// TIA Portal V20 export
// export: Created 2025-12-01T14:56:46.3467956Z, ExportSetting None, DisplayName Totally Integrated Automation Portal, DisplayVersion V20 Update 3, DisplayName TIA Portal Openness, DisplayVersion V20 Update 3, DisplayName TIA Portal Version Control Interface, DisplayVersion V20 Update 3, DisplayName STEP 7 Professional, DisplayVersion V20 Update 3, DisplayName STEP 7 Safety, DisplayVersion V20 Update 2, DisplayName WinCC Basic/Comfort/Advanced, DisplayVersion V20 Update 3, DisplayName WinCC Professional, DisplayVersion V20 Update 3, DisplayName WinCC Unified, DisplayVersion V20 Update 3
FUNCTION_BLOCK "FB263_M_FSS_Maquetas"   // FB263, LAD
TITLE = Control del Ramal de Salidas
{ S7_Optimized_Access := 'FALSE' }
AUTHOR : TE_FSS
NAME : 20160509
VERSION : 3.4
// stored: AutoNumber false, SetENOAutomatically false
   VAR_INPUT
      Mesa : UInt;   // Existe Tension en la Mesa
      Error_Tx : Bool;   // Error en el Tx
      EnTension : Bool;   // Mesa de la FB
      Termico_Tx : Bool;   // Proteccion del Tx
      pHsMx_MQ1 : Bool;   // pHs de la Mesa >> En MQ1
      pHsMx_MQ2 : Bool;   // pHs de la Mesa >> En MQ2
      Avance_Tx : Bool;   // Avance del Tx
      TP1_Arriba : Bool;   // TP1 Arriba. Nota Movimiento E1 >> S3
      TP1_Abajo : Bool;   // TP1 Abajo. Nota Movimiento E1 >> S3
      EnMovimiento_TP1 : Bool;   // En movimiento el TP1
      MQ1_Arriba : Bool;   // MQ1 Arriba >> 1º UT de la Mesa
      MQ1_Abajo : Bool;   // MQ1 Abajo >> 1º UT de la Mesa
      EnMovimiento_MQ1 : Bool;   // MQ1 EnMovimiento >> 1º UT de la Mesa
      MQ2_Arriba : Bool;   // MQ2 Arriba >> 2º UT de la Mesa
      MQ2_Abajo : Bool;   // MQ2 Abajo >> 2º UT de la Mesa
      EnMovimiento_MQ2 : Bool;   // MQ2 EnMovimiento >> 2º UT de la Mesa
      MAnt_DescargaAct : Bool;   // E1 >> Mesa Anterior DescargaAct
      AVTF_MAnt_Mx_MQ1 : Bool;   // E1 >> Mesa Anterior AVTF
      AVTF_MAnt_Mx_MQ1_2 : Bool;   // E1 >> Mesa Anterior AVTF
      P_Mens_MAnt_Mx : Bool;   // E1 >> Mesa Anterior P_Mens
      PTF_Mx_MSig : Bool;   // S3 >> Mesa Siguiente PTF
      FTF_Mx_MSig : Bool;   // S3 >> Mesa Siguiente FTF
      MSig_CargaAct : Bool;
      Mx_ControlUTs : Bool;   // Config >> Control de UT en Mesa
      F_EnvMens_Mx : Bool;   // Fin de Envio de Mensaje
      OrdSal_MQ1 : Bool;   // Orden de Salida de MQ1
      OrdSal_MQ2 : Bool;   // Orden de Salida de MQ2
      OrdSal_MQ1_2 : Bool;   // Orden de Salida de MQ1 y MQ2
      V_CNT_pHsMx : Int := 400;   // Valor de Presencia
      V_CNT_pHsMx_FTF : Int := 200;   // Valor para activar FTF. Nota: < = V_CNT_pHsMx.
      V_CNTSeg_pHsMx : Int := 2000;   // Valor de Seguriadad para Presencia
      V_CNT_ApHsMx : Int := 200;   // Valor de Ausencia
      V_CNTSeg_ApHsMx : Int := 2000;   // Valor de Seguriadad para Ausencia
      V_CNT_Simultaneo : Int := 2000;   // Valor de Simultaneo
      V_EstabilidadCarga : Time := T#200MS;   // Valor de Estabilidad de la Carga
      V_RetardoBajarMAQ : Time := T#200MS;   // Valor de Retardo de Bajada de las Maquetas
      V_TOut_Tx_Mx : Int := 7000;   // TimeOut de Entrada por E1
      V_TOut_TP : Int := 3000;   // TimeOut de Tope
      V_TOut_MQ : Int := 3000;   // TimeOut de Maqueta
      V_CNT_PerdidapHs : Int := 1000;   // CNT de Perdida de pHs
   END_VAR
   VAR_OUTPUT
      P_EnvMens_PMx : Bool;   // Permiso de Enviar Mensaje de Presencia
      P_RecepOK_Mx : Bool;   // Recepcion OK
      PTF_MAnt_Mx : Bool;   // E1 >> Mesa Anterior PTF
      FTF_MAnt_Mx : Bool;   // E1 >> Mesa Anterior FTF
      AVTF_Mx_MSig_MQ1 : Bool;   // S3 >> Mesa Siguiente AVTF
      AVTF_Mx_MSig_MQ2 : Bool;   // S3 >> Mesa Siguiente AVTF
      AVTF_Mx_MSig_MQ1_2 : Bool;   // S3 >> Mesa Siguiente AVTF
      P_Mens_Mx_MSig : Bool;   // S3 >> Mesa Siguiente P_Mens
   END_VAR
   VAR
      Mx_ET00 : Bool;
      Mx_ET01 : Bool;
      Mx_ET02 : Bool;
      Mx_ET06 : Bool;
      Mx_ET07 : Bool;
      Mx_ET08 : Bool;
      Mx_ET09 : Bool;
      Mx_ET10 : Bool;
      Mx_ET11 : Bool;
      Mx_ET12 : Bool;
      Mx_ET110 : Bool;
      Mx_ET111 : Bool;
      Mx_ET50 : Bool;
      Mx_ET51 : Bool;
      Mx_ET150 : Bool;
      Mx_ET151 : Bool;
      SinUTs_EnMesa : Bool;   // Control UTs En Mesa >> Sin UTs
      DoblePeque_EnMesa : Bool;   // Control UTs En Mesa >> Caja Doble Pequeña
      UT01Peque_EnMesa : Bool;   // Control UTs En Mesa >> UT01 Caja Pequeña
      UT02Peque_EnMesa : Bool;   // Control UTs En Mesa >> UT02 Caja Pequeña
      OrdSalida_OK : Bool;   // Control UTs En Mesa >> Validar Orden de Salida
      Selec_Entrada : Bool;   // Select Entrada de Mesa Anterior
      Selec_Salida_MQ1 : Bool;   // Select Salida de MQ1
      Selec_Salida_MQ2 : Bool;   // Select Salida de MQ2
      Selec_Salida_MQ1_2 : Bool;   // Select Salida de MQ1 y MQ2
      AVTF_MAnt_Mx : Bool;   // Interna >> Aviso de Entrada
      AVTF_Mx_MSig : Bool;   // Interna >> Aviso de Salida
      SaliendoCarga : Bool;   // Interna >> Realizando Salida de la Mesa
      PosMQ_OK : Bool;   // Interna >> Pos. de Maquetas OK
      Simultaneo_Mx : Bool;   // Activo Simultaneo E1
      ProtocoloIniciado : Bool;   // Iniciado el Envio del Mensaje de Presencia
      CNT_pHsMx_FTF_OK : Bool;   // Enviar ya FTF
      STAT_EnvMens_PMx : Bool;   // Interna >> Envio del Mensaje de Presencia
      STAT_FTF_MAnt_Mx : Bool;   // Interna >> FTF de MAnt >> Mx
      MA_Subir_MQ1 : Bool;
      MA_Bajar_MQ1 : Bool;
      MA_Subir_MQ2 : Bool;
      MA_Bajar_MQ2 : Bool;
      TMP_EstabilidadCarga { S7_SetPoint := 'True'} : TON_TIME;   // TMP de Estabilidad de la Carga En la Entrada
      TMP_RetardoBajada_MQ1 { S7_SetPoint := 'True'} : TON_TIME;   // TMP de Retardo de Bajada de la MQ1
      TMP_RetardoBajada_MQ2 { S7_SetPoint := 'True'} : TON_TIME;   // TMP de Retardo de Bajada de la MQ2
      CNT_pHsMx { S7_SetPoint := 'True'} : "FB910_CNT_UHS";   // CNT de la Presencia
      CNTSeg_pHsMx { S7_SetPoint := 'True'} : "FB910_CNT_UHS";   // CNT de Seguridad de la Presencia
      CNT_ApHsMx { S7_SetPoint := 'True'} : "FB910_CNT_UHS";   // CNT de la Ausencia
      CNTSeg_ApHsMx { S7_SetPoint := 'True'} : "FB910_CNT_UHS";   // CNT de Seguridad de la Ausencia
      CNT_Simultaneo { S7_SetPoint := 'True'} : "FB910_CNT_UHS";   // CNT de Simultaneo
      TMP_EnTension { S7_SetPoint := 'True'} : "FB910_CNT_UHS";
      TOut_Av_Mx { S7_SetPoint := 'True'} : "FB910_CNT_UHS";   // Time Out de Entrada de E1
      TOut_Subir_TP { S7_SetPoint := 'True'} : "FB910_CNT_UHS";   // Time Out de Subida del TP
      TOut_Bajar_TP { S7_SetPoint := 'True'} : "FB910_CNT_UHS";   // Time Out de Bajada del TP
      TOut_Subir_MQ { S7_SetPoint := 'True'} : "FB910_CNT_UHS";
      TOut_Bajar_MQ { S7_SetPoint := 'True'} : "FB910_CNT_UHS";
      CNT_PerdidapHs { S7_SetPoint := 'True'} : "FB910_CNT_UHS";   // CNT de Perdida de pHs
   END_VAR
   VAR_TEMP
      EstadoZona : "EstadoZona";   // Estado de Zona de la Mesa
      EstadoVI : "EstadosMesa";   // Estado del Vehiculo Inteliguente de la Mesa
      ConfigFB : "UDT_ConfigFB";   // Configuracion de la FB de la Mesa
      V_Protrusion : Int;
      Aux_ET00 : Bool;
   END_VAR
   VAR_TEMP   // added for the SCL form of the ladder/FBD networks
      _w1 : Bool;
   END_VAR
BEGIN

REGION Network 1: INICIALIZAR - Recoger las Variables de Estado de la Mesa
   // Se recoge - Estado_CBx
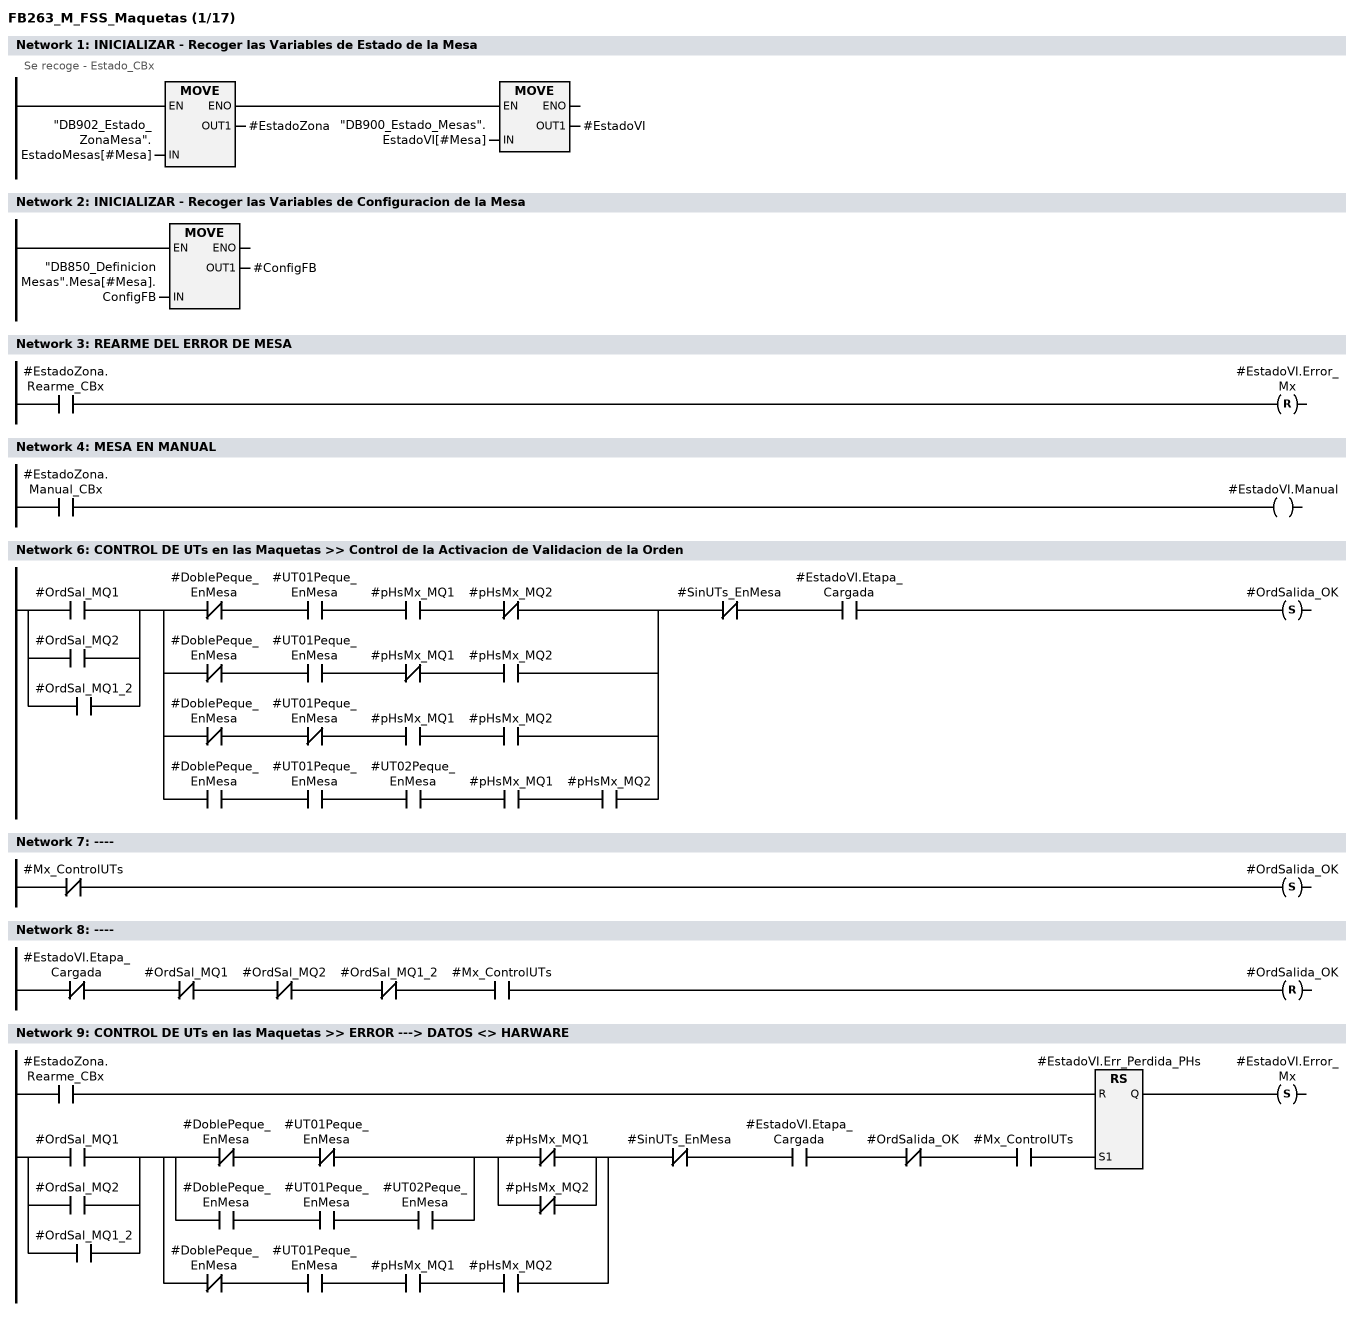
   RUNG wire#powerrail
      Move(in := "DB902_Estado_ZonaMesa".EstadoMesas[#Mesa], out1 => #EstadoZona)
      Move(in := "DB900_Estado_Mesas".EstadoVI[#Mesa], out1 => #EstadoVI)
   END_RUNG
   // the same network as SCL:
   #EstadoZona := "DB902_Estado_ZonaMesa".EstadoMesas[#Mesa];
   #EstadoVI := "DB900_Estado_Mesas".EstadoVI[#Mesa];
END_REGION

REGION Network 2: INICIALIZAR - Recoger las Variables de Configuracion de la Mesa
   RUNG wire#powerrail
      Move(in := "DB850_DefinicionMesas".Mesa[#Mesa].ConfigFB, out1 => #ConfigFB)
   END_RUNG
   // the same network as SCL:
   #ConfigFB := "DB850_DefinicionMesas".Mesa[#Mesa].ConfigFB;
END_REGION

REGION Network 3: REARME DEL ERROR DE MESA
   RUNG wire#powerrail
      Contact( #EstadoZona.Rearme_CBx )
      R_Coil( #EstadoVI.Error_Mx )
   END_RUNG
   // the same network as SCL:
   IF #EstadoZona.Rearme_CBx THEN #EstadoVI.Error_Mx := FALSE; END_IF;
END_REGION

REGION Network 4: MESA EN MANUAL
   RUNG wire#powerrail
      Contact( #EstadoZona.Manual_CBx )
      Coil( #EstadoVI.Manual )
   END_RUNG
   // the same network as SCL:
   #EstadoVI.Manual := #EstadoZona.Manual_CBx;
END_REGION

NETWORK
TITLE = CONTROL DE UTs en las Maquetas >> Recoger datos de las UTs de la Mesa
//////////////////////////////////////////////////////////////////////////////////
/// Recoger datos de las UTs de la Mesa

      CALL  "FC870_MesaSinUT"
      ( Mesa  := #Mesa,
        SinUT := #SinUTs_EnMesa
      );

      CALL  "FC777_TipoCajaPlastico_EnMesa"
      ( Mesa           := #Mesa,
        DosCajas       := #DoblePeque_EnMesa,
        CajaPeque_UT01 := #UT01Peque_EnMesa,
        CajaPeque_UT02 := #UT02Peque_EnMesa
      );



REGION Network 6: CONTROL DE UTs en las Maquetas >> Control de la Activacion de Validacion de la Orden
   RUNG wire#powerrail
      Contact( #OrdSal_MQ1 )
      wire#w1
      I_Contact( #DoblePeque_EnMesa )
      Contact( #UT01Peque_EnMesa )
      Contact( #pHsMx_MQ1 )
      I_Contact( #pHsMx_MQ2 )
      wire#w2
      I_Contact( #SinUTs_EnMesa )
      Contact( #EstadoVI.Etapa_Cargada )
      S_Coil( #OrdSalida_OK )
   END_RUNG
   RUNG wire#powerrail
      Contact( #OrdSal_MQ2 )
   END_RUNG wire#w1
   RUNG wire#powerrail
      Contact( #OrdSal_MQ1_2 )
   END_RUNG wire#w1
   RUNG wire#w1
      I_Contact( #DoblePeque_EnMesa )
      Contact( #UT01Peque_EnMesa )
      I_Contact( #pHsMx_MQ1 )
      Contact( #pHsMx_MQ2 )
   END_RUNG wire#w2
   RUNG wire#w1
      I_Contact( #DoblePeque_EnMesa )
      I_Contact( #UT01Peque_EnMesa )
      Contact( #pHsMx_MQ1 )
      Contact( #pHsMx_MQ2 )
   END_RUNG wire#w2
   RUNG wire#w1
      Contact( #DoblePeque_EnMesa )
      Contact( #UT01Peque_EnMesa )
      Contact( #UT02Peque_EnMesa )
      Contact( #pHsMx_MQ1 )
      Contact( #pHsMx_MQ2 )
   END_RUNG wire#w2
   // the same network as SCL:
   IF (#OrdSal_MQ1 OR #OrdSal_MQ2 OR #OrdSal_MQ1_2) AND ((NOT #DoblePeque_EnMesa AND #UT01Peque_EnMesa AND #pHsMx_MQ1 AND NOT #pHsMx_MQ2) OR (NOT #DoblePeque_EnMesa AND #UT01Peque_EnMesa AND NOT #pHsMx_MQ1 AND #pHsMx_MQ2) OR (NOT #DoblePeque_EnMesa AND NOT #UT01Peque_EnMesa AND #pHsMx_MQ1 AND #pHsMx_MQ2) OR (#DoblePeque_EnMesa AND #UT01Peque_EnMesa AND #UT02Peque_EnMesa AND #pHsMx_MQ1 AND #pHsMx_MQ2)) AND NOT #SinUTs_EnMesa AND #EstadoVI.Etapa_Cargada THEN
       #OrdSalida_OK := TRUE;
   END_IF;
END_REGION

REGION Network 7: ----
   RUNG wire#powerrail
      I_Contact( #Mx_ControlUTs )
      S_Coil( #OrdSalida_OK )
   END_RUNG
   // the same network as SCL:
   IF NOT #Mx_ControlUTs THEN #OrdSalida_OK := TRUE; END_IF;
END_REGION

REGION Network 8: ----
   RUNG wire#powerrail
      I_Contact( #EstadoVI.Etapa_Cargada )
      I_Contact( #OrdSal_MQ1 )
      I_Contact( #OrdSal_MQ2 )
      I_Contact( #OrdSal_MQ1_2 )
      Contact( #Mx_ControlUTs )
      R_Coil( #OrdSalida_OK )
   END_RUNG
   // the same network as SCL:
   IF NOT #EstadoVI.Etapa_Cargada AND NOT #OrdSal_MQ1 AND NOT #OrdSal_MQ2 AND NOT #OrdSal_MQ1_2 AND #Mx_ControlUTs THEN
       #OrdSalida_OK := FALSE;
   END_IF;
END_REGION

REGION Network 9: CONTROL DE UTs en las Maquetas >> ERROR ---> DATOS <> HARWARE
   RUNG wire#powerrail
      Contact( #EstadoZona.Rearme_CBx )
      S_RS(operand := #EstadoVI.Err_Perdida_PHs, s1 := wire#w4)
      S_Coil( #EstadoVI.Error_Mx )
   END_RUNG
   RUNG wire#powerrail
      Contact( #OrdSal_MQ1 )
      wire#w1
      I_Contact( #DoblePeque_EnMesa )
      I_Contact( #UT01Peque_EnMesa )
      wire#w2
      I_Contact( #pHsMx_MQ1 )
      wire#w3
      I_Contact( #SinUTs_EnMesa )
      Contact( #EstadoVI.Etapa_Cargada )
      I_Contact( #OrdSalida_OK )
      Contact( #Mx_ControlUTs )
   END_RUNG wire#w4
   RUNG wire#powerrail
      Contact( #OrdSal_MQ2 )
   END_RUNG wire#w1
   RUNG wire#powerrail
      Contact( #OrdSal_MQ1_2 )
   END_RUNG wire#w1
   RUNG wire#w1
      Contact( #DoblePeque_EnMesa )
      Contact( #UT01Peque_EnMesa )
      Contact( #UT02Peque_EnMesa )
   END_RUNG wire#w2
   RUNG wire#w2
      I_Contact( #pHsMx_MQ2 )
   END_RUNG wire#w3
   RUNG wire#w1
      I_Contact( #DoblePeque_EnMesa )
      Contact( #UT01Peque_EnMesa )
      Contact( #pHsMx_MQ1 )
      Contact( #pHsMx_MQ2 )
   END_RUNG wire#w3
   // the same network as SCL:
   IF #EstadoZona.Rearme_CBx THEN
       #EstadoVI.Err_Perdida_PHs := FALSE;   // RS flip-flop
   END_IF;
   IF (#OrdSal_MQ1 OR #OrdSal_MQ2 OR #OrdSal_MQ1_2) AND ((((NOT #DoblePeque_EnMesa AND NOT #UT01Peque_EnMesa) OR (#DoblePeque_EnMesa AND #UT01Peque_EnMesa AND #UT02Peque_EnMesa)) AND (NOT #pHsMx_MQ1 OR NOT #pHsMx_MQ2)) OR (NOT #DoblePeque_EnMesa AND #UT01Peque_EnMesa AND #pHsMx_MQ1 AND #pHsMx_MQ2)) AND NOT #SinUTs_EnMesa AND #EstadoVI.Etapa_Cargada AND NOT #OrdSalida_OK AND #Mx_ControlUTs THEN
       #EstadoVI.Err_Perdida_PHs := TRUE;
   END_IF;
   IF #EstadoVI.Err_Perdida_PHs THEN #EstadoVI.Error_Mx := TRUE; END_IF;
END_REGION

REGION Network 10: VARIABLES AUXILIARES - Aviso de Entrada - AVTF_MAnt_Mx
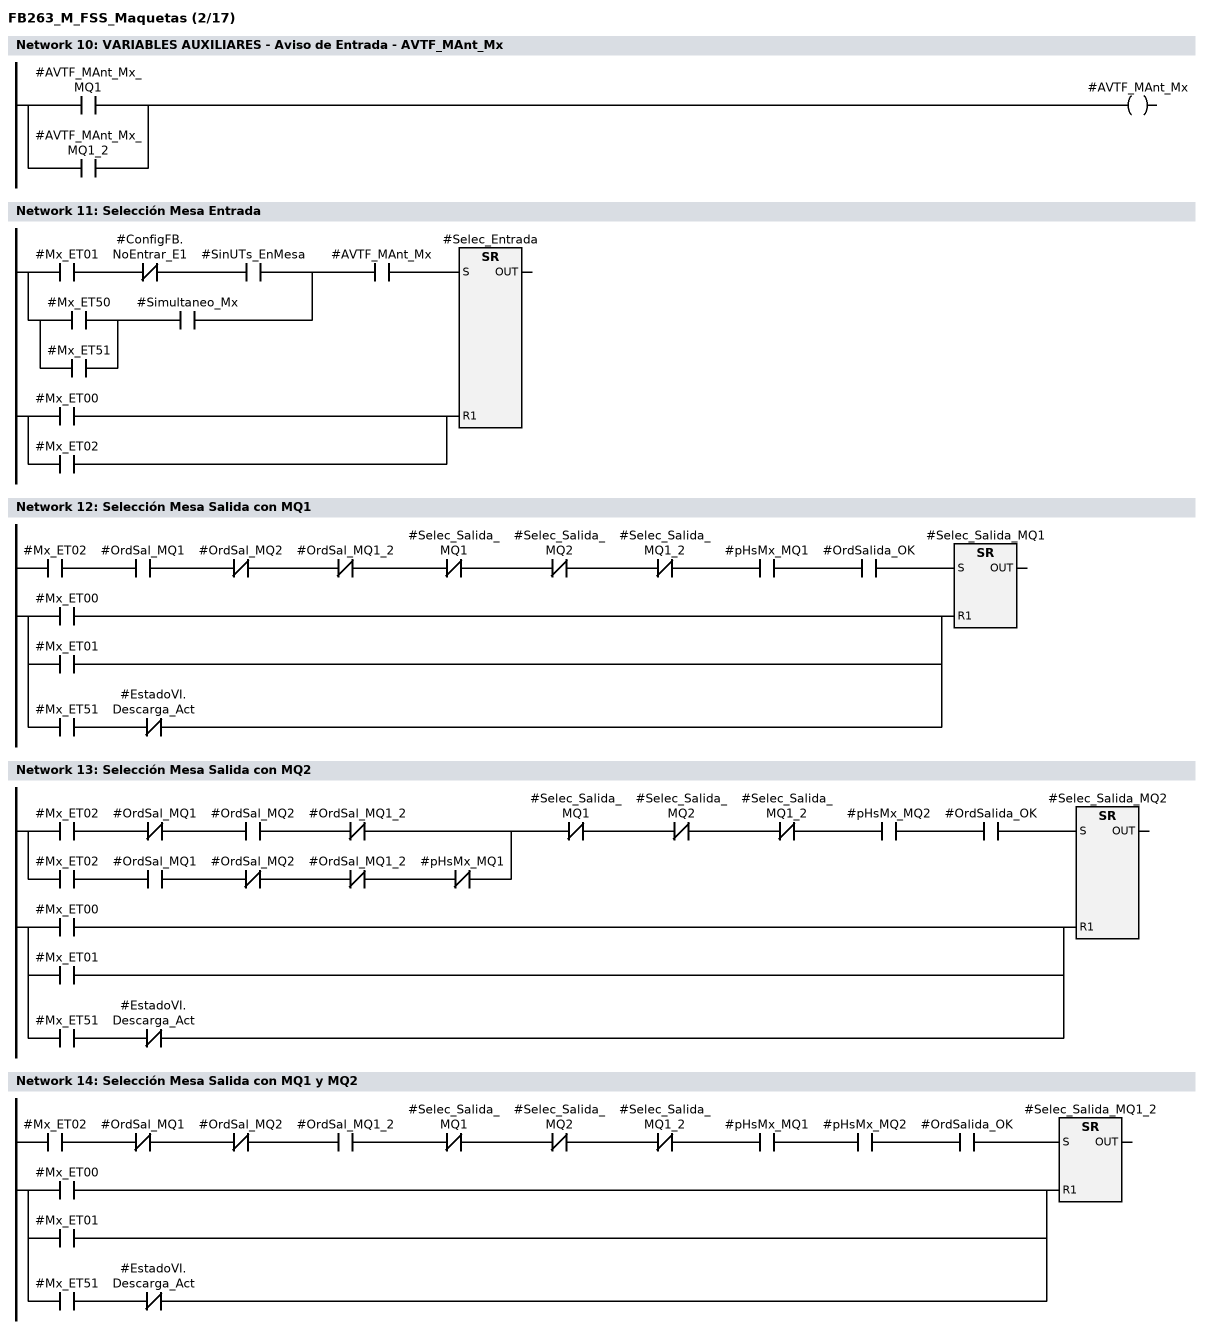
   RUNG wire#powerrail
      Contact( #AVTF_MAnt_Mx_MQ1 )
      wire#w1
      Coil( #AVTF_MAnt_Mx )
   END_RUNG
   RUNG wire#powerrail
      Contact( #AVTF_MAnt_Mx_MQ1_2 )
   END_RUNG wire#w1
   // the same network as SCL:
   #AVTF_MAnt_Mx := #AVTF_MAnt_Mx_MQ1 OR #AVTF_MAnt_Mx_MQ1_2;
END_REGION

REGION Network 11: Selección Mesa Entrada
   RUNG wire#powerrail
      Contact( #Mx_ET01 )
      I_Contact( #ConfigFB.NoEntrar_E1 )
      Contact( #SinUTs_EnMesa )
      wire#w1
      Contact( #AVTF_MAnt_Mx )
      S_SR(operand := #Selec_Entrada, r1 := wire#w3)
   END_RUNG
   RUNG wire#powerrail
      Contact( #Mx_ET50 )
      wire#w2
      Contact( #Simultaneo_Mx )
   END_RUNG wire#w1
   RUNG wire#powerrail
      Contact( #Mx_ET51 )
   END_RUNG wire#w2
   RUNG wire#powerrail
      Contact( #Mx_ET00 )
   END_RUNG wire#w3
   RUNG wire#powerrail
      Contact( #Mx_ET02 )
   END_RUNG wire#w3
   // the same network as SCL:
   IF ((#Mx_ET01 AND NOT #ConfigFB.NoEntrar_E1 AND #SinUTs_EnMesa) OR ((#Mx_ET50 OR #Mx_ET51) AND #Simultaneo_Mx)) AND #AVTF_MAnt_Mx THEN
       #Selec_Entrada := TRUE;   // SR flip-flop
   END_IF;
   IF #Mx_ET00 OR #Mx_ET02 THEN #Selec_Entrada := FALSE; END_IF;
END_REGION

REGION Network 12: Selección Mesa Salida con MQ1
   RUNG wire#powerrail
      Contact( #Mx_ET02 )
      Contact( #OrdSal_MQ1 )
      I_Contact( #OrdSal_MQ2 )
      I_Contact( #OrdSal_MQ1_2 )
      I_Contact( #Selec_Salida_MQ1 )
      I_Contact( #Selec_Salida_MQ2 )
      I_Contact( #Selec_Salida_MQ1_2 )
      Contact( #pHsMx_MQ1 )
      Contact( #OrdSalida_OK )
      S_SR(operand := #Selec_Salida_MQ1, r1 := wire#w1)
   END_RUNG
   RUNG wire#powerrail
      Contact( #Mx_ET00 )
   END_RUNG wire#w1
   RUNG wire#powerrail
      Contact( #Mx_ET01 )
   END_RUNG wire#w1
   RUNG wire#powerrail
      Contact( #Mx_ET51 )
      I_Contact( #EstadoVI.Descarga_Act )
   END_RUNG wire#w1
   // the same network as SCL:
   IF #Mx_ET02 AND #OrdSal_MQ1 AND NOT #OrdSal_MQ2 AND NOT #OrdSal_MQ1_2 AND NOT #Selec_Salida_MQ1 AND NOT #Selec_Salida_MQ2 AND NOT #Selec_Salida_MQ1_2 AND #pHsMx_MQ1 AND #OrdSalida_OK THEN
       #Selec_Salida_MQ1 := TRUE;   // SR flip-flop
   END_IF;
   IF #Mx_ET00 OR #Mx_ET01 OR (#Mx_ET51 AND NOT #EstadoVI.Descarga_Act) THEN
       #Selec_Salida_MQ1 := FALSE;
   END_IF;
END_REGION

REGION Network 13: Selección Mesa Salida con MQ2
   RUNG wire#powerrail
      Contact( #Mx_ET02 )
      I_Contact( #OrdSal_MQ1 )
      Contact( #OrdSal_MQ2 )
      I_Contact( #OrdSal_MQ1_2 )
      wire#w1
      I_Contact( #Selec_Salida_MQ1 )
      I_Contact( #Selec_Salida_MQ2 )
      I_Contact( #Selec_Salida_MQ1_2 )
      Contact( #pHsMx_MQ2 )
      Contact( #OrdSalida_OK )
      S_SR(operand := #Selec_Salida_MQ2, r1 := wire#w2)
   END_RUNG
   RUNG wire#powerrail
      Contact( #Mx_ET02 )
      Contact( #OrdSal_MQ1 )
      I_Contact( #OrdSal_MQ2 )
      I_Contact( #OrdSal_MQ1_2 )
      I_Contact( #pHsMx_MQ1 )
   END_RUNG wire#w1
   RUNG wire#powerrail
      Contact( #Mx_ET00 )
   END_RUNG wire#w2
   RUNG wire#powerrail
      Contact( #Mx_ET01 )
   END_RUNG wire#w2
   RUNG wire#powerrail
      Contact( #Mx_ET51 )
      I_Contact( #EstadoVI.Descarga_Act )
   END_RUNG wire#w2
   // the same network as SCL:
   IF ((#Mx_ET02 AND NOT #OrdSal_MQ1 AND #OrdSal_MQ2 AND NOT #OrdSal_MQ1_2) OR (#Mx_ET02 AND #OrdSal_MQ1 AND NOT #OrdSal_MQ2 AND NOT #OrdSal_MQ1_2 AND NOT #pHsMx_MQ1)) AND NOT #Selec_Salida_MQ1 AND NOT #Selec_Salida_MQ2 AND NOT #Selec_Salida_MQ1_2 AND #pHsMx_MQ2 AND #OrdSalida_OK THEN
       #Selec_Salida_MQ2 := TRUE;   // SR flip-flop
   END_IF;
   IF #Mx_ET00 OR #Mx_ET01 OR (#Mx_ET51 AND NOT #EstadoVI.Descarga_Act) THEN
       #Selec_Salida_MQ2 := FALSE;
   END_IF;
END_REGION

REGION Network 14: Selección Mesa Salida con MQ1 y MQ2
   RUNG wire#powerrail
      Contact( #Mx_ET02 )
      I_Contact( #OrdSal_MQ1 )
      I_Contact( #OrdSal_MQ2 )
      Contact( #OrdSal_MQ1_2 )
      I_Contact( #Selec_Salida_MQ1 )
      I_Contact( #Selec_Salida_MQ2 )
      I_Contact( #Selec_Salida_MQ1_2 )
      Contact( #pHsMx_MQ1 )
      Contact( #pHsMx_MQ2 )
      Contact( #OrdSalida_OK )
      S_SR(operand := #Selec_Salida_MQ1_2, r1 := wire#w1)
   END_RUNG
   RUNG wire#powerrail
      Contact( #Mx_ET00 )
   END_RUNG wire#w1
   RUNG wire#powerrail
      Contact( #Mx_ET01 )
   END_RUNG wire#w1
   RUNG wire#powerrail
      Contact( #Mx_ET51 )
      I_Contact( #EstadoVI.Descarga_Act )
   END_RUNG wire#w1
   // the same network as SCL:
   IF #Mx_ET02 AND NOT #OrdSal_MQ1 AND NOT #OrdSal_MQ2 AND #OrdSal_MQ1_2 AND NOT #Selec_Salida_MQ1 AND NOT #Selec_Salida_MQ2 AND NOT #Selec_Salida_MQ1_2 AND #pHsMx_MQ1 AND #pHsMx_MQ2 AND #OrdSalida_OK THEN
       #Selec_Salida_MQ1_2 := TRUE;   // SR flip-flop
   END_IF;
   IF #Mx_ET00 OR #Mx_ET01 OR (#Mx_ET51 AND NOT #EstadoVI.Descarga_Act) THEN
       #Selec_Salida_MQ1_2 := FALSE;
   END_IF;
END_REGION

REGION Network 15: VARIABLES AUXILIARES - Saliendo Carga de la Mesa
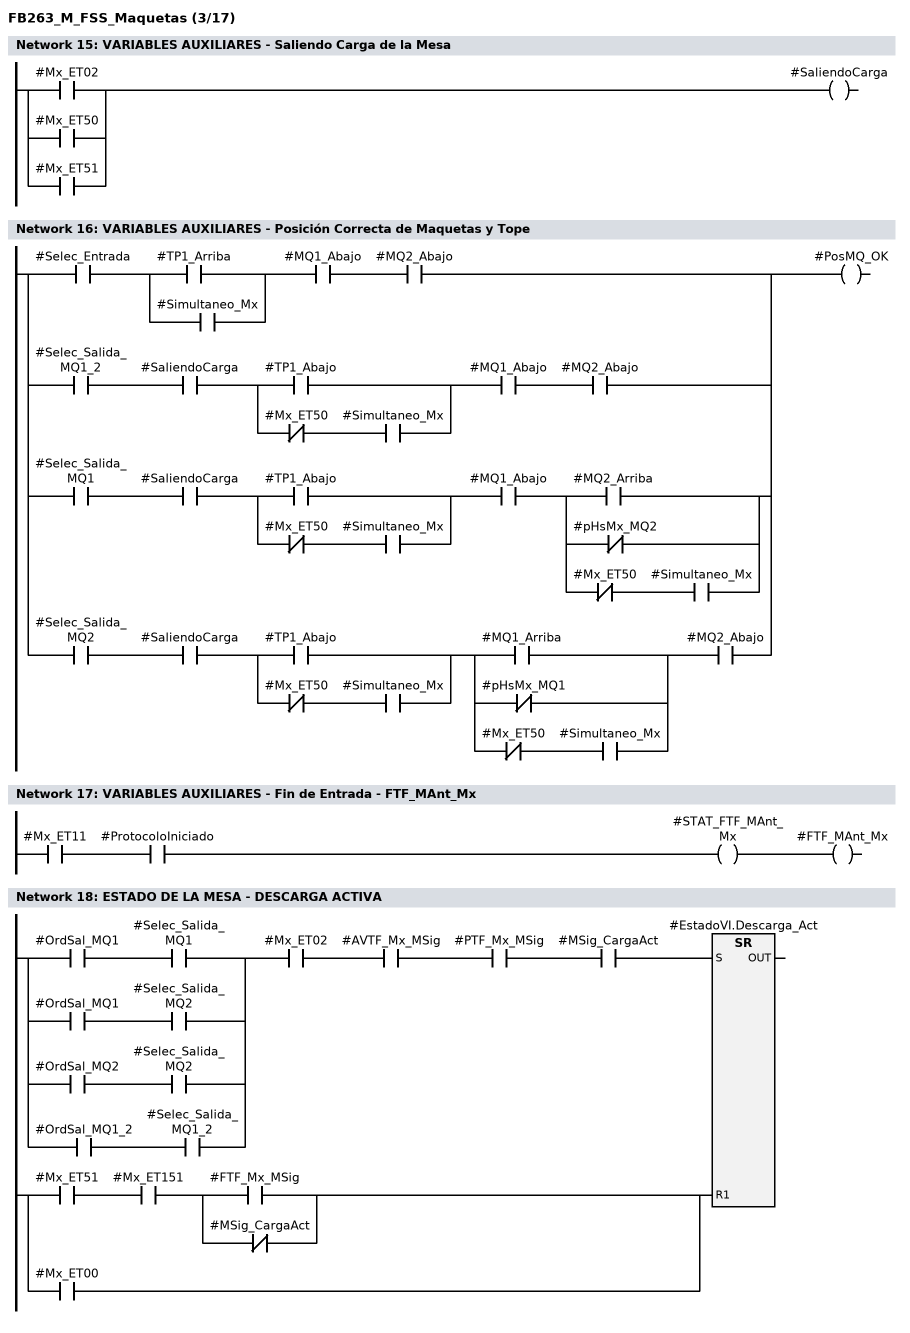
   RUNG wire#powerrail
      Contact( #Mx_ET02 )
      wire#w1
      Coil( #SaliendoCarga )
   END_RUNG
   RUNG wire#powerrail
      Contact( #Mx_ET50 )
   END_RUNG wire#w1
   RUNG wire#powerrail
      Contact( #Mx_ET51 )
   END_RUNG wire#w1
   // the same network as SCL:
   #SaliendoCarga := #Mx_ET02 OR #Mx_ET50 OR #Mx_ET51;
END_REGION

REGION Network 16: VARIABLES AUXILIARES - Posición Correcta de Maquetas y Tope
   RUNG wire#powerrail
      Contact( #Selec_Entrada )
      wire#w1
      Contact( #TP1_Arriba )
      wire#w2
      Contact( #MQ1_Abajo )
      Contact( #MQ2_Abajo )
      wire#w3
      Coil( #PosMQ_OK )
   END_RUNG
   RUNG wire#w1
      Contact( #Simultaneo_Mx )
   END_RUNG wire#w2
   RUNG wire#powerrail
      Contact( #Selec_Salida_MQ1_2 )
      Contact( #SaliendoCarga )
      wire#w4
      Contact( #TP1_Abajo )
      wire#w5
      Contact( #MQ1_Abajo )
      Contact( #MQ2_Abajo )
   END_RUNG wire#w3
   RUNG wire#w4
      I_Contact( #Mx_ET50 )
      Contact( #Simultaneo_Mx )
   END_RUNG wire#w5
   RUNG wire#powerrail
      Contact( #Selec_Salida_MQ1 )
      Contact( #SaliendoCarga )
      wire#w6
      Contact( #TP1_Abajo )
      wire#w7
      Contact( #MQ1_Abajo )
      wire#w8
      Contact( #MQ2_Arriba )
   END_RUNG wire#w3
   RUNG wire#w6
      I_Contact( #Mx_ET50 )
      Contact( #Simultaneo_Mx )
   END_RUNG wire#w7
   RUNG wire#w8
      I_Contact( #pHsMx_MQ2 )
   END_RUNG wire#w3
   RUNG wire#w8
      I_Contact( #Mx_ET50 )
      Contact( #Simultaneo_Mx )
   END_RUNG wire#w3
   RUNG wire#powerrail
      Contact( #Selec_Salida_MQ2 )
      Contact( #SaliendoCarga )
      wire#w9
      Contact( #TP1_Abajo )
      wire#w10
      Contact( #MQ1_Arriba )
      wire#w11
      Contact( #MQ2_Abajo )
   END_RUNG wire#w3
   RUNG wire#w9
      I_Contact( #Mx_ET50 )
      Contact( #Simultaneo_Mx )
   END_RUNG wire#w10
   RUNG wire#w10
      I_Contact( #pHsMx_MQ1 )
   END_RUNG wire#w11
   RUNG wire#w10
      I_Contact( #Mx_ET50 )
      Contact( #Simultaneo_Mx )
   END_RUNG wire#w11
   // the same network as SCL:
   #PosMQ_OK := (#Selec_Entrada AND (#TP1_Arriba OR #Simultaneo_Mx) AND #MQ1_Abajo AND #MQ2_Abajo) OR (#Selec_Salida_MQ1_2 AND #SaliendoCarga AND (#TP1_Abajo OR (NOT #Mx_ET50 AND #Simultaneo_Mx)) AND #MQ1_Abajo AND #MQ2_Abajo) OR (#Selec_Salida_MQ1 AND #SaliendoCarga AND (#TP1_Abajo OR (NOT #Mx_ET50 AND #Simultaneo_Mx)) AND #MQ1_Abajo AND (#MQ2_Arriba OR NOT #pHsMx_MQ2 OR (NOT #Mx_ET50 AND #Simultaneo_Mx))) OR (#Selec_Salida_MQ2 AND #SaliendoCarga AND (#TP1_Abajo OR (NOT #Mx_ET50 AND #Simultaneo_Mx)) AND (#MQ1_Arriba OR NOT #pHsMx_MQ1 OR (NOT #Mx_ET50 AND #Simultaneo_Mx)) AND #MQ2_Abajo);
END_REGION

REGION Network 17: VARIABLES AUXILIARES - Fin de Entrada - FTF_MAnt_Mx
   RUNG wire#powerrail
      Contact( #Mx_ET11 )
      Contact( #ProtocoloIniciado )
      Coil( #STAT_FTF_MAnt_Mx )
      Coil( #FTF_MAnt_Mx )
   END_RUNG
   // the same network as SCL:
   #STAT_FTF_MAnt_Mx := #Mx_ET11 AND #ProtocoloIniciado;
   #FTF_MAnt_Mx := #STAT_FTF_MAnt_Mx;
END_REGION

REGION Network 18: ESTADO DE LA MESA - DESCARGA ACTIVA
   RUNG wire#powerrail
      Contact( #OrdSal_MQ1 )
      Contact( #Selec_Salida_MQ1 )
      wire#w1
      Contact( #Mx_ET02 )
      Contact( #AVTF_Mx_MSig )
      Contact( #PTF_Mx_MSig )
      Contact( #MSig_CargaAct )
      S_SR(operand := #EstadoVI.Descarga_Act, r1 := wire#w3)
   END_RUNG
   RUNG wire#powerrail
      Contact( #OrdSal_MQ1 )
      Contact( #Selec_Salida_MQ2 )
   END_RUNG wire#w1
   RUNG wire#powerrail
      Contact( #OrdSal_MQ2 )
      Contact( #Selec_Salida_MQ2 )
   END_RUNG wire#w1
   RUNG wire#powerrail
      Contact( #OrdSal_MQ1_2 )
      Contact( #Selec_Salida_MQ1_2 )
   END_RUNG wire#w1
   RUNG wire#powerrail
      Contact( #Mx_ET51 )
      Contact( #Mx_ET151 )
      wire#w2
      Contact( #FTF_Mx_MSig )
   END_RUNG wire#w3
   RUNG wire#w2
      I_Contact( #MSig_CargaAct )
   END_RUNG wire#w3
   RUNG wire#powerrail
      Contact( #Mx_ET00 )
   END_RUNG wire#w3
   // the same network as SCL:
   IF ((#OrdSal_MQ1 AND #Selec_Salida_MQ1) OR (#OrdSal_MQ1 AND #Selec_Salida_MQ2) OR (#OrdSal_MQ2 AND #Selec_Salida_MQ2) OR (#OrdSal_MQ1_2 AND #Selec_Salida_MQ1_2)) AND #Mx_ET02 AND #AVTF_Mx_MSig AND #PTF_Mx_MSig AND #MSig_CargaAct THEN
       #EstadoVI.Descarga_Act := TRUE;   // SR flip-flop
   END_IF;
   IF (#Mx_ET51 AND #Mx_ET151 AND (#FTF_Mx_MSig OR NOT #MSig_CargaAct)) OR #Mx_ET00 THEN
       #EstadoVI.Descarga_Act := FALSE;
   END_IF;
END_REGION

REGION Network 19: ET151 - CONTROL DE SALIDA DE CARGA - PROTOCOLO
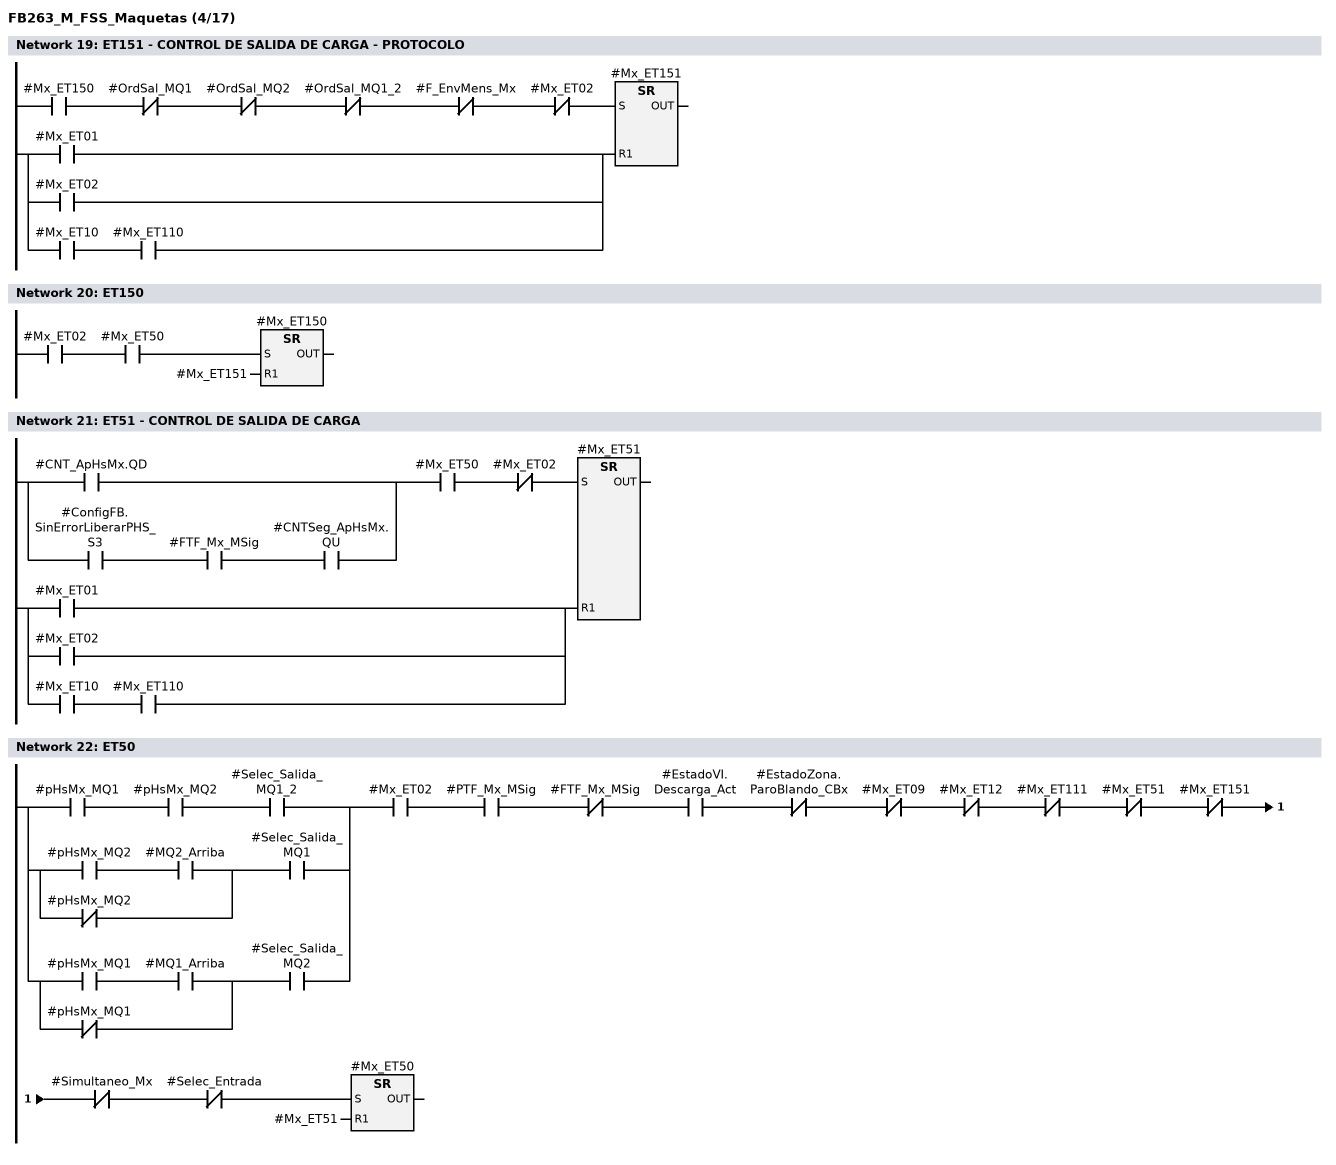
   RUNG wire#powerrail
      Contact( #Mx_ET150 )
      I_Contact( #OrdSal_MQ1 )
      I_Contact( #OrdSal_MQ2 )
      I_Contact( #OrdSal_MQ1_2 )
      I_Contact( #F_EnvMens_Mx )
      I_Contact( #Mx_ET02 )
      S_SR(operand := #Mx_ET151, r1 := wire#w1)
   END_RUNG
   RUNG wire#powerrail
      Contact( #Mx_ET01 )
   END_RUNG wire#w1
   RUNG wire#powerrail
      Contact( #Mx_ET02 )
   END_RUNG wire#w1
   RUNG wire#powerrail
      Contact( #Mx_ET10 )
      Contact( #Mx_ET110 )
   END_RUNG wire#w1
   // the same network as SCL:
   IF #Mx_ET150 AND NOT #OrdSal_MQ1 AND NOT #OrdSal_MQ2 AND NOT #OrdSal_MQ1_2 AND NOT #F_EnvMens_Mx AND NOT #Mx_ET02 THEN
       #Mx_ET151 := TRUE;   // SR flip-flop
   END_IF;
   IF #Mx_ET01 OR #Mx_ET02 OR (#Mx_ET10 AND #Mx_ET110) THEN #Mx_ET151 := FALSE; END_IF;
END_REGION

REGION Network 20: ET150
   RUNG wire#powerrail
      Contact( #Mx_ET02 )
      Contact( #Mx_ET50 )
      S_SR(operand := #Mx_ET150, r1 := #Mx_ET151)
   END_RUNG
   // the same network as SCL:
   IF #Mx_ET02 AND #Mx_ET50 THEN
       #Mx_ET150 := TRUE;   // SR flip-flop
   END_IF;
   IF #Mx_ET151 THEN #Mx_ET150 := FALSE; END_IF;
END_REGION

REGION Network 21: ET51 - CONTROL DE SALIDA DE CARGA
   RUNG wire#powerrail
      Contact( #CNT_ApHsMx.QD )
      wire#w1
      Contact( #Mx_ET50 )
      I_Contact( #Mx_ET02 )
      S_SR(operand := #Mx_ET51, r1 := wire#w2)
   END_RUNG
   RUNG wire#powerrail
      Contact( #ConfigFB.SinErrorLiberarPHS_S3 )
      Contact( #FTF_Mx_MSig )
      Contact( #CNTSeg_ApHsMx.QU )
   END_RUNG wire#w1
   RUNG wire#powerrail
      Contact( #Mx_ET01 )
   END_RUNG wire#w2
   RUNG wire#powerrail
      Contact( #Mx_ET02 )
   END_RUNG wire#w2
   RUNG wire#powerrail
      Contact( #Mx_ET10 )
      Contact( #Mx_ET110 )
   END_RUNG wire#w2
   // the same network as SCL:
   IF (#CNT_ApHsMx.QD OR (#ConfigFB.SinErrorLiberarPHS_S3 AND #FTF_Mx_MSig AND #CNTSeg_ApHsMx.QU)) AND #Mx_ET50 AND NOT #Mx_ET02 THEN
       #Mx_ET51 := TRUE;   // SR flip-flop
   END_IF;
   IF #Mx_ET01 OR #Mx_ET02 OR (#Mx_ET10 AND #Mx_ET110) THEN #Mx_ET51 := FALSE; END_IF;
END_REGION

REGION Network 22: ET50
   RUNG wire#powerrail
      Contact( #pHsMx_MQ1 )
      Contact( #pHsMx_MQ2 )
      Contact( #Selec_Salida_MQ1_2 )
      wire#w1
      Contact( #Mx_ET02 )
      Contact( #PTF_Mx_MSig )
      I_Contact( #FTF_Mx_MSig )
      Contact( #EstadoVI.Descarga_Act )
      I_Contact( #EstadoZona.ParoBlando_CBx )
      I_Contact( #Mx_ET09 )
      I_Contact( #Mx_ET12 )
      I_Contact( #Mx_ET111 )
      I_Contact( #Mx_ET51 )
      I_Contact( #Mx_ET151 )
      I_Contact( #Simultaneo_Mx )
      I_Contact( #Selec_Entrada )
      S_SR(operand := #Mx_ET50, r1 := #Mx_ET51)
   END_RUNG
   RUNG wire#powerrail
      Contact( #pHsMx_MQ2 )
      Contact( #MQ2_Arriba )
      wire#w2
      Contact( #Selec_Salida_MQ1 )
   END_RUNG wire#w1
   RUNG wire#powerrail
      I_Contact( #pHsMx_MQ2 )
   END_RUNG wire#w2
   RUNG wire#powerrail
      Contact( #pHsMx_MQ1 )
      Contact( #MQ1_Arriba )
      wire#w3
      Contact( #Selec_Salida_MQ2 )
   END_RUNG wire#w1
   RUNG wire#powerrail
      I_Contact( #pHsMx_MQ1 )
   END_RUNG wire#w3
   // the same network as SCL:
   IF ((#pHsMx_MQ1 AND #pHsMx_MQ2 AND #Selec_Salida_MQ1_2) OR (((#pHsMx_MQ2 AND #MQ2_Arriba) OR NOT #pHsMx_MQ2) AND #Selec_Salida_MQ1) OR (((#pHsMx_MQ1 AND #MQ1_Arriba) OR NOT #pHsMx_MQ1) AND #Selec_Salida_MQ2)) AND #Mx_ET02 AND #PTF_Mx_MSig AND NOT #FTF_Mx_MSig AND #EstadoVI.Descarga_Act AND NOT #EstadoZona.ParoBlando_CBx AND NOT #Mx_ET09 AND NOT #Mx_ET12 AND NOT #Mx_ET111 AND NOT #Mx_ET51 AND NOT #Mx_ET151 AND NOT #Simultaneo_Mx AND NOT #Selec_Entrada THEN
       #Mx_ET50 := TRUE;   // SR flip-flop
   END_IF;
   IF #Mx_ET51 THEN #Mx_ET50 := FALSE; END_IF;
END_REGION

REGION Network 23: ET02 - ESTADO DE REPOSO CARGADA
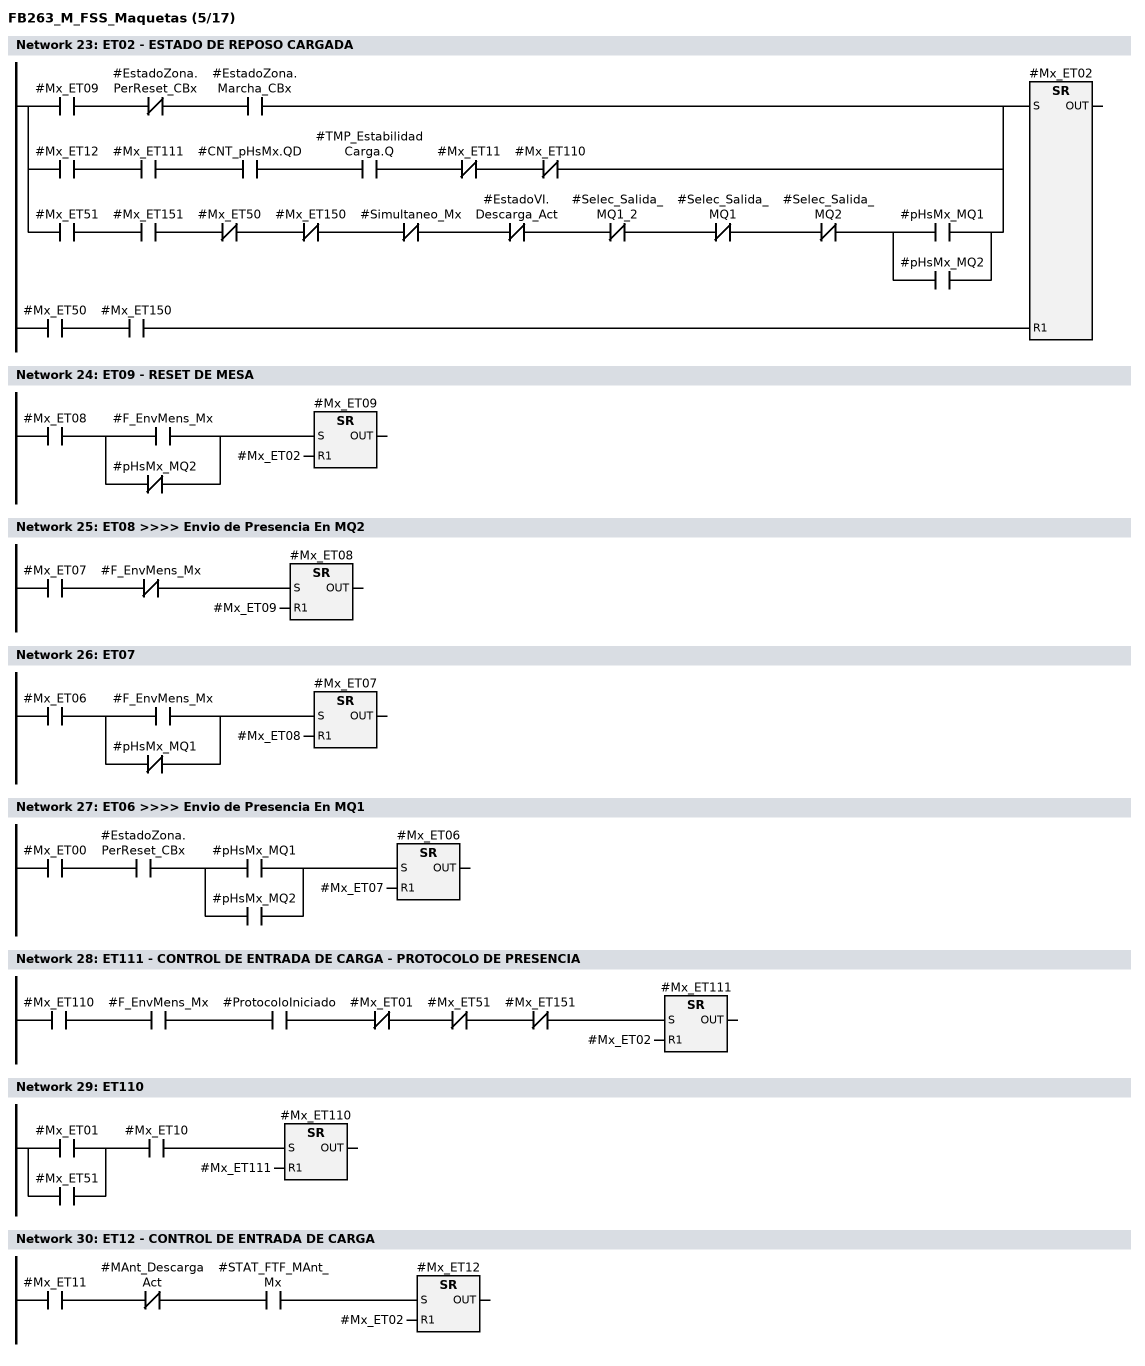
   RUNG wire#powerrail
      Contact( #Mx_ET09 )
      I_Contact( #EstadoZona.PerReset_CBx )
      Contact( #EstadoZona.Marcha_CBx )
      wire#w1
      S_SR(operand := #Mx_ET02, r1 := wire#w3)
   END_RUNG
   RUNG wire#powerrail
      Contact( #Mx_ET12 )
      Contact( #Mx_ET111 )
      Contact( #CNT_pHsMx.QD )
      Contact( #TMP_EstabilidadCarga.Q )
      I_Contact( #Mx_ET11 )
      I_Contact( #Mx_ET110 )
   END_RUNG wire#w1
   RUNG wire#powerrail
      Contact( #Mx_ET51 )
      Contact( #Mx_ET151 )
      I_Contact( #Mx_ET50 )
      I_Contact( #Mx_ET150 )
      I_Contact( #Simultaneo_Mx )
      I_Contact( #EstadoVI.Descarga_Act )
      I_Contact( #Selec_Salida_MQ1_2 )
      I_Contact( #Selec_Salida_MQ1 )
      I_Contact( #Selec_Salida_MQ2 )
      wire#w2
      Contact( #pHsMx_MQ1 )
   END_RUNG wire#w1
   RUNG wire#w2
      Contact( #pHsMx_MQ2 )
   END_RUNG wire#w1
   RUNG wire#powerrail
      Contact( #Mx_ET50 )
      Contact( #Mx_ET150 )
   END_RUNG wire#w3
   // the same network as SCL:
   IF (#Mx_ET09 AND NOT #EstadoZona.PerReset_CBx AND #EstadoZona.Marcha_CBx) OR (#Mx_ET12 AND #Mx_ET111 AND #CNT_pHsMx.QD AND #TMP_EstabilidadCarga.Q AND NOT #Mx_ET11 AND NOT #Mx_ET110) OR (#Mx_ET51 AND #Mx_ET151 AND NOT #Mx_ET50 AND NOT #Mx_ET150 AND NOT #Simultaneo_Mx AND NOT #EstadoVI.Descarga_Act AND NOT #Selec_Salida_MQ1_2 AND NOT #Selec_Salida_MQ1 AND NOT #Selec_Salida_MQ2 AND (#pHsMx_MQ1 OR #pHsMx_MQ2)) THEN
       #Mx_ET02 := TRUE;   // SR flip-flop
   END_IF;
   IF #Mx_ET50 AND #Mx_ET150 THEN #Mx_ET02 := FALSE; END_IF;
END_REGION

REGION Network 24: ET09 - RESET DE MESA
   RUNG wire#powerrail
      Contact( #Mx_ET08 )
      wire#w1
      Contact( #F_EnvMens_Mx )
      wire#w2
      S_SR(operand := #Mx_ET09, r1 := #Mx_ET02)
   END_RUNG
   RUNG wire#w1
      I_Contact( #pHsMx_MQ2 )
   END_RUNG wire#w2
   // the same network as SCL:
   IF #Mx_ET08 AND (#F_EnvMens_Mx OR NOT #pHsMx_MQ2) THEN
       #Mx_ET09 := TRUE;   // SR flip-flop
   END_IF;
   IF #Mx_ET02 THEN #Mx_ET09 := FALSE; END_IF;
END_REGION

REGION Network 25: ET08 >>>> Envio de Presencia En MQ2
   RUNG wire#powerrail
      Contact( #Mx_ET07 )
      I_Contact( #F_EnvMens_Mx )
      S_SR(operand := #Mx_ET08, r1 := #Mx_ET09)
   END_RUNG
   // the same network as SCL:
   IF #Mx_ET07 AND NOT #F_EnvMens_Mx THEN
       #Mx_ET08 := TRUE;   // SR flip-flop
   END_IF;
   IF #Mx_ET09 THEN #Mx_ET08 := FALSE; END_IF;
END_REGION

REGION Network 26: ET07
   RUNG wire#powerrail
      Contact( #Mx_ET06 )
      wire#w1
      Contact( #F_EnvMens_Mx )
      wire#w2
      S_SR(operand := #Mx_ET07, r1 := #Mx_ET08)
   END_RUNG
   RUNG wire#w1
      I_Contact( #pHsMx_MQ1 )
   END_RUNG wire#w2
   // the same network as SCL:
   IF #Mx_ET06 AND (#F_EnvMens_Mx OR NOT #pHsMx_MQ1) THEN
       #Mx_ET07 := TRUE;   // SR flip-flop
   END_IF;
   IF #Mx_ET08 THEN #Mx_ET07 := FALSE; END_IF;
END_REGION

REGION Network 27: ET06 >>>> Envio de Presencia En MQ1
   RUNG wire#powerrail
      Contact( #Mx_ET00 )
      Contact( #EstadoZona.PerReset_CBx )
      wire#w1
      Contact( #pHsMx_MQ1 )
      wire#w2
      S_SR(operand := #Mx_ET06, r1 := #Mx_ET07)
   END_RUNG
   RUNG wire#w1
      Contact( #pHsMx_MQ2 )
   END_RUNG wire#w2
   // the same network as SCL:
   IF #Mx_ET00 AND #EstadoZona.PerReset_CBx AND (#pHsMx_MQ1 OR #pHsMx_MQ2) THEN
       #Mx_ET06 := TRUE;   // SR flip-flop
   END_IF;
   IF #Mx_ET07 THEN #Mx_ET06 := FALSE; END_IF;
END_REGION

REGION Network 28: ET111 - CONTROL DE ENTRADA DE CARGA - PROTOCOLO DE PRESENCIA
   RUNG wire#powerrail
      Contact( #Mx_ET110 )
      Contact( #F_EnvMens_Mx )
      Contact( #ProtocoloIniciado )
      I_Contact( #Mx_ET01 )
      I_Contact( #Mx_ET51 )
      I_Contact( #Mx_ET151 )
      S_SR(operand := #Mx_ET111, r1 := #Mx_ET02)
   END_RUNG
   // the same network as SCL:
   IF #Mx_ET110 AND #F_EnvMens_Mx AND #ProtocoloIniciado AND NOT #Mx_ET01 AND NOT #Mx_ET51 AND NOT #Mx_ET151 THEN
       #Mx_ET111 := TRUE;   // SR flip-flop
   END_IF;
   IF #Mx_ET02 THEN #Mx_ET111 := FALSE; END_IF;
END_REGION

REGION Network 29: ET110
   RUNG wire#powerrail
      Contact( #Mx_ET01 )
      wire#w1
      Contact( #Mx_ET10 )
      S_SR(operand := #Mx_ET110, r1 := #Mx_ET111)
   END_RUNG
   RUNG wire#powerrail
      Contact( #Mx_ET51 )
   END_RUNG wire#w1
   // the same network as SCL:
   IF (#Mx_ET01 OR #Mx_ET51) AND #Mx_ET10 THEN
       #Mx_ET110 := TRUE;   // SR flip-flop
   END_IF;
   IF #Mx_ET111 THEN #Mx_ET110 := FALSE; END_IF;
END_REGION

REGION Network 30: ET12 - CONTROL DE ENTRADA DE CARGA
   RUNG wire#powerrail
      Contact( #Mx_ET11 )
      I_Contact( #MAnt_DescargaAct )
      Contact( #STAT_FTF_MAnt_Mx )
      S_SR(operand := #Mx_ET12, r1 := #Mx_ET02)
   END_RUNG
   // the same network as SCL:
   IF #Mx_ET11 AND NOT #MAnt_DescargaAct AND #STAT_FTF_MAnt_Mx THEN
       #Mx_ET12 := TRUE;   // SR flip-flop
   END_IF;
   IF #Mx_ET02 THEN #Mx_ET12 := FALSE; END_IF;
END_REGION

REGION Network 31: ET11
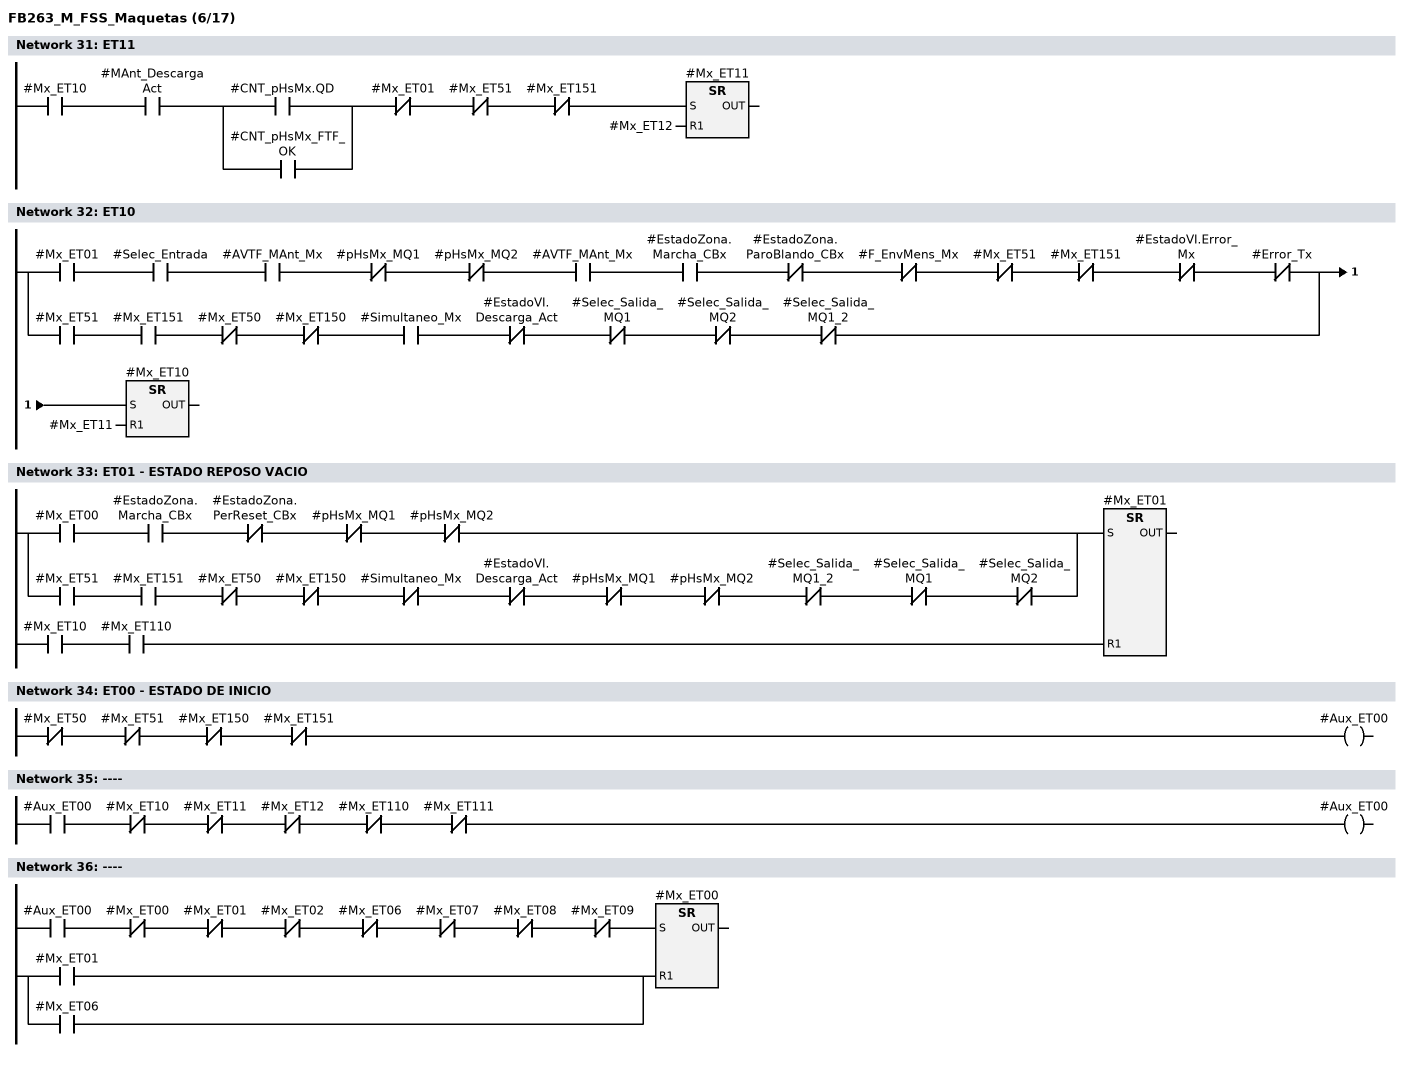
   RUNG wire#powerrail
      Contact( #Mx_ET10 )
      Contact( #MAnt_DescargaAct )
      wire#w1
      Contact( #CNT_pHsMx.QD )
      wire#w2
      I_Contact( #Mx_ET01 )
      I_Contact( #Mx_ET51 )
      I_Contact( #Mx_ET151 )
      S_SR(operand := #Mx_ET11, r1 := #Mx_ET12)
   END_RUNG
   RUNG wire#w1
      Contact( #CNT_pHsMx_FTF_OK )
   END_RUNG wire#w2
   // the same network as SCL:
   IF #Mx_ET10 AND #MAnt_DescargaAct AND (#CNT_pHsMx.QD OR #CNT_pHsMx_FTF_OK) AND NOT #Mx_ET01 AND NOT #Mx_ET51 AND NOT #Mx_ET151 THEN
       #Mx_ET11 := TRUE;   // SR flip-flop
   END_IF;
   IF #Mx_ET12 THEN #Mx_ET11 := FALSE; END_IF;
END_REGION

REGION Network 32: ET10
   RUNG wire#powerrail
      Contact( #Mx_ET01 )
      Contact( #Selec_Entrada )
      Contact( #AVTF_MAnt_Mx )
      I_Contact( #pHsMx_MQ1 )
      I_Contact( #pHsMx_MQ2 )
      Contact( #AVTF_MAnt_Mx )
      Contact( #EstadoZona.Marcha_CBx )
      I_Contact( #EstadoZona.ParoBlando_CBx )
      I_Contact( #F_EnvMens_Mx )
      I_Contact( #Mx_ET51 )
      I_Contact( #Mx_ET151 )
      I_Contact( #EstadoVI.Error_Mx )
      I_Contact( #Error_Tx )
      wire#w1
      S_SR(operand := #Mx_ET10, r1 := #Mx_ET11)
   END_RUNG
   RUNG wire#powerrail
      Contact( #Mx_ET51 )
      Contact( #Mx_ET151 )
      I_Contact( #Mx_ET50 )
      I_Contact( #Mx_ET150 )
      Contact( #Simultaneo_Mx )
      I_Contact( #EstadoVI.Descarga_Act )
      I_Contact( #Selec_Salida_MQ1 )
      I_Contact( #Selec_Salida_MQ2 )
      I_Contact( #Selec_Salida_MQ1_2 )
   END_RUNG wire#w1
   // the same network as SCL:
   IF (#Mx_ET01 AND #Selec_Entrada AND #AVTF_MAnt_Mx AND NOT #pHsMx_MQ1 AND NOT #pHsMx_MQ2 AND #AVTF_MAnt_Mx AND #EstadoZona.Marcha_CBx AND NOT #EstadoZona.ParoBlando_CBx AND NOT #F_EnvMens_Mx AND NOT #Mx_ET51 AND NOT #Mx_ET151 AND NOT #EstadoVI.Error_Mx AND NOT #Error_Tx) OR (#Mx_ET51 AND #Mx_ET151 AND NOT #Mx_ET50 AND NOT #Mx_ET150 AND #Simultaneo_Mx AND NOT #EstadoVI.Descarga_Act AND NOT #Selec_Salida_MQ1 AND NOT #Selec_Salida_MQ2 AND NOT #Selec_Salida_MQ1_2) THEN
       #Mx_ET10 := TRUE;   // SR flip-flop
   END_IF;
   IF #Mx_ET11 THEN #Mx_ET10 := FALSE; END_IF;
END_REGION

REGION Network 33: ET01 - ESTADO REPOSO VACIO
   RUNG wire#powerrail
      Contact( #Mx_ET00 )
      Contact( #EstadoZona.Marcha_CBx )
      I_Contact( #EstadoZona.PerReset_CBx )
      I_Contact( #pHsMx_MQ1 )
      I_Contact( #pHsMx_MQ2 )
      wire#w1
      S_SR(operand := #Mx_ET01, r1 := wire#w2)
   END_RUNG
   RUNG wire#powerrail
      Contact( #Mx_ET51 )
      Contact( #Mx_ET151 )
      I_Contact( #Mx_ET50 )
      I_Contact( #Mx_ET150 )
      I_Contact( #Simultaneo_Mx )
      I_Contact( #EstadoVI.Descarga_Act )
      I_Contact( #pHsMx_MQ1 )
      I_Contact( #pHsMx_MQ2 )
      I_Contact( #Selec_Salida_MQ1_2 )
      I_Contact( #Selec_Salida_MQ1 )
      I_Contact( #Selec_Salida_MQ2 )
   END_RUNG wire#w1
   RUNG wire#powerrail
      Contact( #Mx_ET10 )
      Contact( #Mx_ET110 )
   END_RUNG wire#w2
   // the same network as SCL:
   IF (#Mx_ET00 AND #EstadoZona.Marcha_CBx AND NOT #EstadoZona.PerReset_CBx AND NOT #pHsMx_MQ1 AND NOT #pHsMx_MQ2) OR (#Mx_ET51 AND #Mx_ET151 AND NOT #Mx_ET50 AND NOT #Mx_ET150 AND NOT #Simultaneo_Mx AND NOT #EstadoVI.Descarga_Act AND NOT #pHsMx_MQ1 AND NOT #pHsMx_MQ2 AND NOT #Selec_Salida_MQ1_2 AND NOT #Selec_Salida_MQ1 AND NOT #Selec_Salida_MQ2) THEN
       #Mx_ET01 := TRUE;   // SR flip-flop
   END_IF;
   IF #Mx_ET10 AND #Mx_ET110 THEN #Mx_ET01 := FALSE; END_IF;
END_REGION

REGION Network 34: ET00 - ESTADO DE INICIO
   RUNG wire#powerrail
      I_Contact( #Mx_ET50 )
      I_Contact( #Mx_ET51 )
      I_Contact( #Mx_ET150 )
      I_Contact( #Mx_ET151 )
      Coil( #Aux_ET00 )
   END_RUNG
   // the same network as SCL:
   #Aux_ET00 := NOT #Mx_ET50 AND NOT #Mx_ET51 AND NOT #Mx_ET150 AND NOT #Mx_ET151;
END_REGION

REGION Network 35: ----
   RUNG wire#powerrail
      Contact( #Aux_ET00 )
      I_Contact( #Mx_ET10 )
      I_Contact( #Mx_ET11 )
      I_Contact( #Mx_ET12 )
      I_Contact( #Mx_ET110 )
      I_Contact( #Mx_ET111 )
      Coil( #Aux_ET00 )
   END_RUNG
   // the same network as SCL:
   #Aux_ET00 := #Aux_ET00 AND NOT #Mx_ET10 AND NOT #Mx_ET11 AND NOT #Mx_ET12 AND NOT #Mx_ET110 AND NOT #Mx_ET111;
END_REGION

REGION Network 36: ----
   RUNG wire#powerrail
      Contact( #Aux_ET00 )
      I_Contact( #Mx_ET00 )
      I_Contact( #Mx_ET01 )
      I_Contact( #Mx_ET02 )
      I_Contact( #Mx_ET06 )
      I_Contact( #Mx_ET07 )
      I_Contact( #Mx_ET08 )
      I_Contact( #Mx_ET09 )
      S_SR(operand := #Mx_ET00, r1 := wire#w1)
   END_RUNG
   RUNG wire#powerrail
      Contact( #Mx_ET01 )
   END_RUNG wire#w1
   RUNG wire#powerrail
      Contact( #Mx_ET06 )
   END_RUNG wire#w1
   // the same network as SCL:
   IF #Aux_ET00 AND NOT #Mx_ET00 AND NOT #Mx_ET01 AND NOT #Mx_ET02 AND NOT #Mx_ET06 AND NOT #Mx_ET07 AND NOT #Mx_ET08 AND NOT #Mx_ET09 THEN
       #Mx_ET00 := TRUE;   // SR flip-flop
   END_IF;
   IF #Mx_ET01 OR #Mx_ET06 THEN #Mx_ET00 := FALSE; END_IF;
END_REGION

REGION Network 37: CONTADOR DE SEGURIDAD DE PRESENCIA - CNTSeg_pHsMx
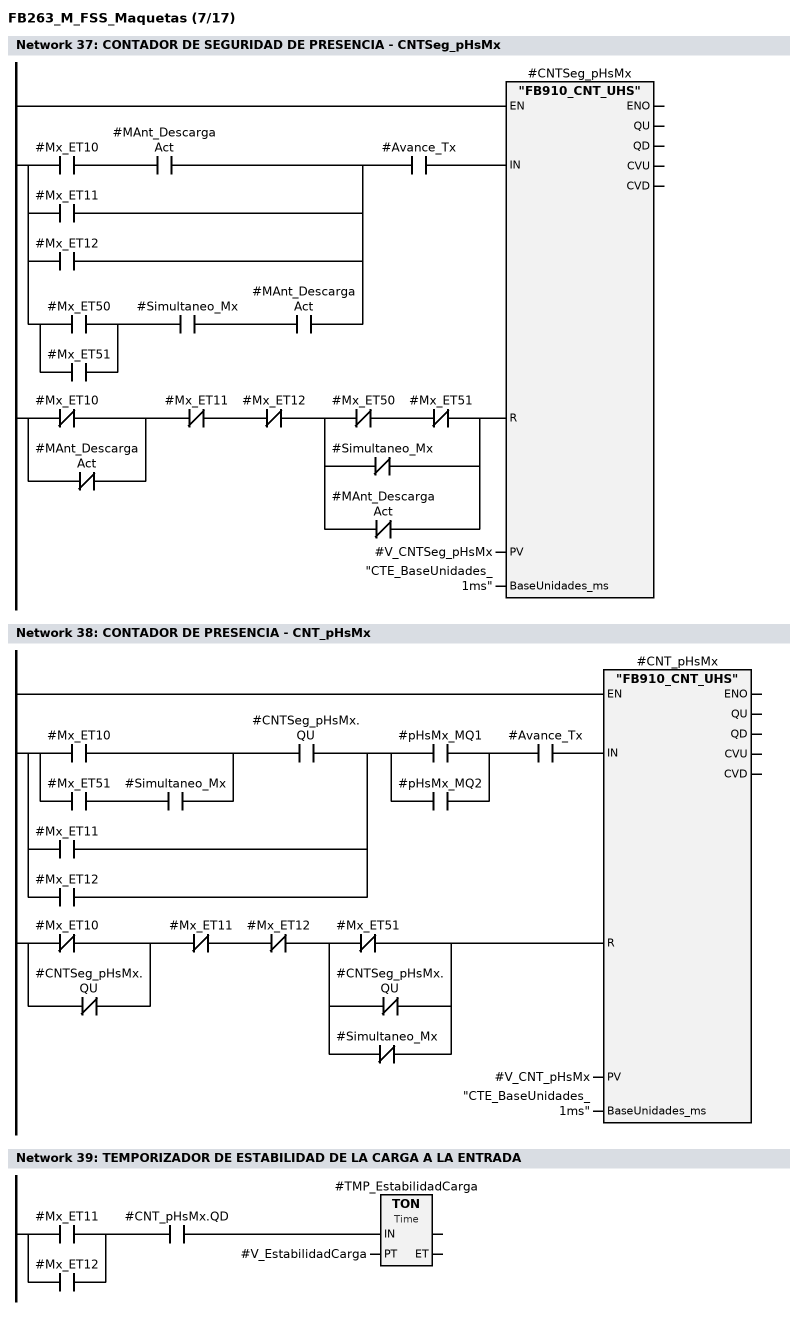
   RUNG wire#powerrail
      #CNTSeg_pHsMx(IN := wire#w3, R := wire#w6, PV := #V_CNTSeg_pHsMx, BaseUnidades_ms := "CTE_BaseUnidades_1ms", QU =>, QD =>, CVU =>, CVD =>)
   END_RUNG
   RUNG wire#powerrail
      Contact( #Mx_ET10 )
      Contact( #MAnt_DescargaAct )
      wire#w1
      Contact( #Avance_Tx )
   END_RUNG wire#w3
   RUNG wire#powerrail
      Contact( #Mx_ET11 )
   END_RUNG wire#w1
   RUNG wire#powerrail
      Contact( #Mx_ET12 )
   END_RUNG wire#w1
   RUNG wire#powerrail
      Contact( #Mx_ET50 )
      wire#w2
      Contact( #Simultaneo_Mx )
      Contact( #MAnt_DescargaAct )
   END_RUNG wire#w1
   RUNG wire#powerrail
      Contact( #Mx_ET51 )
   END_RUNG wire#w2
   RUNG wire#powerrail
      I_Contact( #Mx_ET10 )
      wire#w4
      I_Contact( #Mx_ET11 )
      I_Contact( #Mx_ET12 )
      wire#w5
      I_Contact( #Mx_ET50 )
      I_Contact( #Mx_ET51 )
   END_RUNG wire#w6
   RUNG wire#powerrail
      I_Contact( #MAnt_DescargaAct )
   END_RUNG wire#w4
   RUNG wire#w5
      I_Contact( #Simultaneo_Mx )
   END_RUNG wire#w6
   RUNG wire#w5
      I_Contact( #MAnt_DescargaAct )
   END_RUNG wire#w6
   // the same network as SCL:
   #CNTSeg_pHsMx(IN := ((#Mx_ET10 AND #MAnt_DescargaAct) OR #Mx_ET11 OR #Mx_ET12 OR ((#Mx_ET50 OR #Mx_ET51) AND #Simultaneo_Mx AND #MAnt_DescargaAct)) AND #Avance_Tx,   // "FB910_CNT_UHS"
                 R := (NOT #Mx_ET10 OR NOT #MAnt_DescargaAct) AND NOT #Mx_ET11 AND NOT #Mx_ET12 AND ((NOT #Mx_ET50 AND NOT #Mx_ET51) OR NOT #Simultaneo_Mx OR NOT #MAnt_DescargaAct),
                 PV := #V_CNTSeg_pHsMx,
                 BaseUnidades_ms := "CTE_BaseUnidades_1ms");
END_REGION

REGION Network 38: CONTADOR DE PRESENCIA - CNT_pHsMx
   RUNG wire#powerrail
      #CNT_pHsMx(IN := wire#w4, R := wire#w7, PV := #V_CNT_pHsMx, BaseUnidades_ms := "CTE_BaseUnidades_1ms", QU =>, QD =>, CVU =>, CVD =>)
   END_RUNG
   RUNG wire#powerrail
      Contact( #Mx_ET10 )
      wire#w1
      Contact( #CNTSeg_pHsMx.QU )
      wire#w2
      Contact( #pHsMx_MQ1 )
      wire#w3
      Contact( #Avance_Tx )
   END_RUNG wire#w4
   RUNG wire#powerrail
      Contact( #Mx_ET51 )
      Contact( #Simultaneo_Mx )
   END_RUNG wire#w1
   RUNG wire#powerrail
      Contact( #Mx_ET11 )
   END_RUNG wire#w2
   RUNG wire#powerrail
      Contact( #Mx_ET12 )
   END_RUNG wire#w2
   RUNG wire#w2
      Contact( #pHsMx_MQ2 )
   END_RUNG wire#w3
   RUNG wire#powerrail
      I_Contact( #Mx_ET10 )
      wire#w5
      I_Contact( #Mx_ET11 )
      I_Contact( #Mx_ET12 )
      wire#w6
      I_Contact( #Mx_ET51 )
   END_RUNG wire#w7
   RUNG wire#powerrail
      I_Contact( #CNTSeg_pHsMx.QU )
   END_RUNG wire#w5
   RUNG wire#w6
      I_Contact( #CNTSeg_pHsMx.QU )
   END_RUNG wire#w7
   RUNG wire#w6
      I_Contact( #Simultaneo_Mx )
   END_RUNG wire#w7
   // the same network as SCL:
   #CNT_pHsMx(IN := (((#Mx_ET10 OR (#Mx_ET51 AND #Simultaneo_Mx)) AND #CNTSeg_pHsMx.QU) OR #Mx_ET11 OR #Mx_ET12) AND (#pHsMx_MQ1 OR #pHsMx_MQ2) AND #Avance_Tx,   // "FB910_CNT_UHS"
              R := (NOT #Mx_ET10 OR NOT #CNTSeg_pHsMx.QU) AND NOT #Mx_ET11 AND NOT #Mx_ET12 AND (NOT #Mx_ET51 OR NOT #CNTSeg_pHsMx.QU OR NOT #Simultaneo_Mx),
              PV := #V_CNT_pHsMx,
              BaseUnidades_ms := "CTE_BaseUnidades_1ms");
END_REGION

REGION Network 39: TEMPORIZADOR DE ESTABILIDAD DE LA CARGA A LA ENTRADA
   RUNG wire#powerrail
      Contact( #Mx_ET11 )
      wire#w1
      Contact( #CNT_pHsMx.QD )
      { S7_Templates := "time_type := Time" } #TMP_EstabilidadCarga.TON(pt := #V_EstabilidadCarga, et =>)
   END_RUNG
   RUNG wire#powerrail
      Contact( #Mx_ET12 )
   END_RUNG wire#w1
   // the same network as SCL:
   #TMP_EstabilidadCarga(IN := (#Mx_ET11 OR #Mx_ET12) AND #CNT_pHsMx.QD, PT := #V_EstabilidadCarga);   // TON
END_REGION

REGION Network 40: DETERMINA PASO ET10 - ET11 (Nota: Control de Tiempo para dar el FTF a la Mesa Anterior)
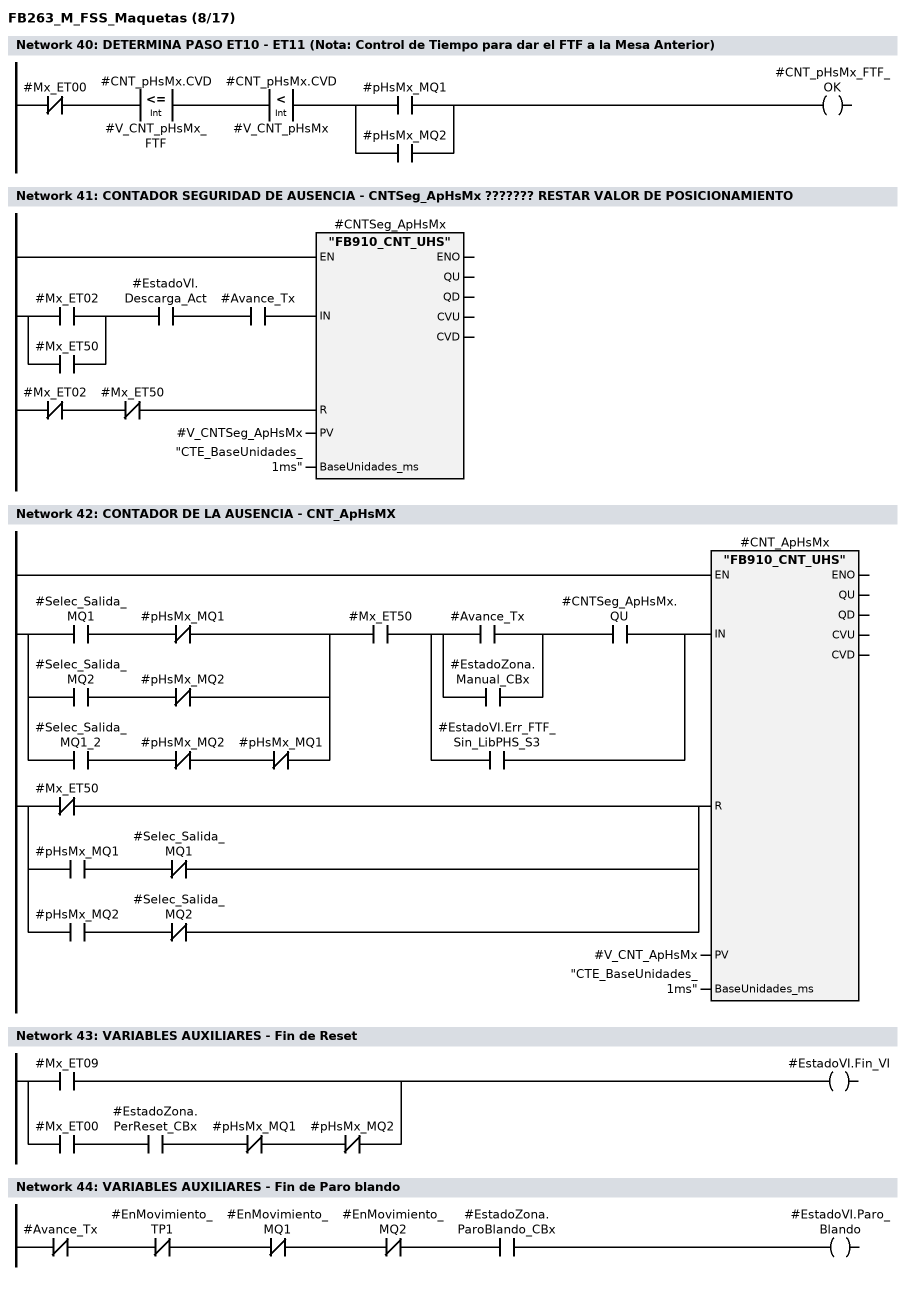
   RUNG wire#powerrail
      I_Contact( #Mx_ET00 )
      { S7_Templates := "SrcType := Int" } LE_Contact(in1 := #CNT_pHsMx.CVD, in2 := #V_CNT_pHsMx_FTF)
      { S7_Templates := "SrcType := Int" } LT_Contact(in1 := #CNT_pHsMx.CVD, in2 := #V_CNT_pHsMx)
      wire#w1
      Contact( #pHsMx_MQ1 )
      wire#w2
      Coil( #CNT_pHsMx_FTF_OK )
   END_RUNG
   RUNG wire#w1
      Contact( #pHsMx_MQ2 )
   END_RUNG wire#w2
   // the same network as SCL:
   #CNT_pHsMx_FTF_OK := NOT #Mx_ET00 AND (#CNT_pHsMx.CVD <= #V_CNT_pHsMx_FTF) AND (#CNT_pHsMx.CVD < #V_CNT_pHsMx) AND (#pHsMx_MQ1 OR #pHsMx_MQ2);
END_REGION

REGION Network 41: CONTADOR SEGURIDAD DE AUSENCIA - CNTSeg_ApHsMx ??????? RESTAR VALOR DE POSICIONAMIENTO
   RUNG wire#powerrail
      #CNTSeg_ApHsMx(IN := wire#w2, R := wire#w3, PV := #V_CNTSeg_ApHsMx, BaseUnidades_ms := "CTE_BaseUnidades_1ms", QU =>, QD =>, CVU =>, CVD =>)
   END_RUNG
   RUNG wire#powerrail
      Contact( #Mx_ET02 )
      wire#w1
      Contact( #EstadoVI.Descarga_Act )
      Contact( #Avance_Tx )
   END_RUNG wire#w2
   RUNG wire#powerrail
      Contact( #Mx_ET50 )
   END_RUNG wire#w1
   RUNG wire#powerrail
      I_Contact( #Mx_ET02 )
      I_Contact( #Mx_ET50 )
   END_RUNG wire#w3
   // the same network as SCL:
   #CNTSeg_ApHsMx(IN := (#Mx_ET02 OR #Mx_ET50) AND #EstadoVI.Descarga_Act AND #Avance_Tx,   // "FB910_CNT_UHS"
                  R := NOT #Mx_ET02 AND NOT #Mx_ET50,
                  PV := #V_CNTSeg_ApHsMx,
                  BaseUnidades_ms := "CTE_BaseUnidades_1ms");
END_REGION

REGION Network 42: CONTADOR DE LA AUSENCIA - CNT_ApHsMX
   RUNG wire#powerrail
      #CNT_ApHsMx(IN := wire#w4, R := wire#w5, PV := #V_CNT_ApHsMx, BaseUnidades_ms := "CTE_BaseUnidades_1ms", QU =>, QD =>, CVU =>, CVD =>)
   END_RUNG
   RUNG wire#powerrail
      Contact( #Selec_Salida_MQ1 )
      I_Contact( #pHsMx_MQ1 )
      wire#w1
      Contact( #Mx_ET50 )
      wire#w2
      Contact( #Avance_Tx )
      wire#w3
      Contact( #CNTSeg_ApHsMx.QU )
   END_RUNG wire#w4
   RUNG wire#powerrail
      Contact( #Selec_Salida_MQ2 )
      I_Contact( #pHsMx_MQ2 )
   END_RUNG wire#w1
   RUNG wire#powerrail
      Contact( #Selec_Salida_MQ1_2 )
      I_Contact( #pHsMx_MQ2 )
      I_Contact( #pHsMx_MQ1 )
   END_RUNG wire#w1
   RUNG wire#w2
      Contact( #EstadoZona.Manual_CBx )
   END_RUNG wire#w3
   RUNG wire#w2
      Contact( #EstadoVI.Err_FTF_Sin_LibPHS_S3 )
   END_RUNG wire#w4
   RUNG wire#powerrail
      I_Contact( #Mx_ET50 )
   END_RUNG wire#w5
   RUNG wire#powerrail
      Contact( #pHsMx_MQ1 )
      I_Contact( #Selec_Salida_MQ1 )
   END_RUNG wire#w5
   RUNG wire#powerrail
      Contact( #pHsMx_MQ2 )
      I_Contact( #Selec_Salida_MQ2 )
   END_RUNG wire#w5
   // the same network as SCL:
   #CNT_ApHsMx(IN := ((#Selec_Salida_MQ1 AND NOT #pHsMx_MQ1) OR (#Selec_Salida_MQ2 AND NOT #pHsMx_MQ2) OR (#Selec_Salida_MQ1_2 AND NOT #pHsMx_MQ2 AND NOT #pHsMx_MQ1)) AND #Mx_ET50 AND (((#Avance_Tx OR #EstadoZona.Manual_CBx) AND #CNTSeg_ApHsMx.QU) OR #EstadoVI.Err_FTF_Sin_LibPHS_S3),   // "FB910_CNT_UHS"
               R := NOT #Mx_ET50 OR (#pHsMx_MQ1 AND NOT #Selec_Salida_MQ1) OR (#pHsMx_MQ2 AND NOT #Selec_Salida_MQ2),
               PV := #V_CNT_ApHsMx,
               BaseUnidades_ms := "CTE_BaseUnidades_1ms");
END_REGION

REGION Network 43: VARIABLES AUXILIARES - Fin de Reset
   RUNG wire#powerrail
      Contact( #Mx_ET09 )
      wire#w1
      Coil( #EstadoVI.Fin_VI )
   END_RUNG
   RUNG wire#powerrail
      Contact( #Mx_ET00 )
      Contact( #EstadoZona.PerReset_CBx )
      I_Contact( #pHsMx_MQ1 )
      I_Contact( #pHsMx_MQ2 )
   END_RUNG wire#w1
   // the same network as SCL:
   #EstadoVI.Fin_VI := #Mx_ET09 OR (#Mx_ET00 AND #EstadoZona.PerReset_CBx AND NOT #pHsMx_MQ1 AND NOT #pHsMx_MQ2);
END_REGION

REGION Network 44: VARIABLES AUXILIARES - Fin de Paro blando
   RUNG wire#powerrail
      I_Contact( #Avance_Tx )
      I_Contact( #EnMovimiento_TP1 )
      I_Contact( #EnMovimiento_MQ1 )
      I_Contact( #EnMovimiento_MQ2 )
      Contact( #EstadoZona.ParoBlando_CBx )
      Coil( #EstadoVI.Paro_Blando )
   END_RUNG
   // the same network as SCL:
   #EstadoVI.Paro_Blando := NOT #Avance_Tx AND NOT #EnMovimiento_TP1 AND NOT #EnMovimiento_MQ1 AND NOT #EnMovimiento_MQ2 AND #EstadoZona.ParoBlando_CBx;
END_REGION

REGION Network 45: VARIABLES AUXILIARES - Permiso de Entrada - PTF_MAnt_Mx
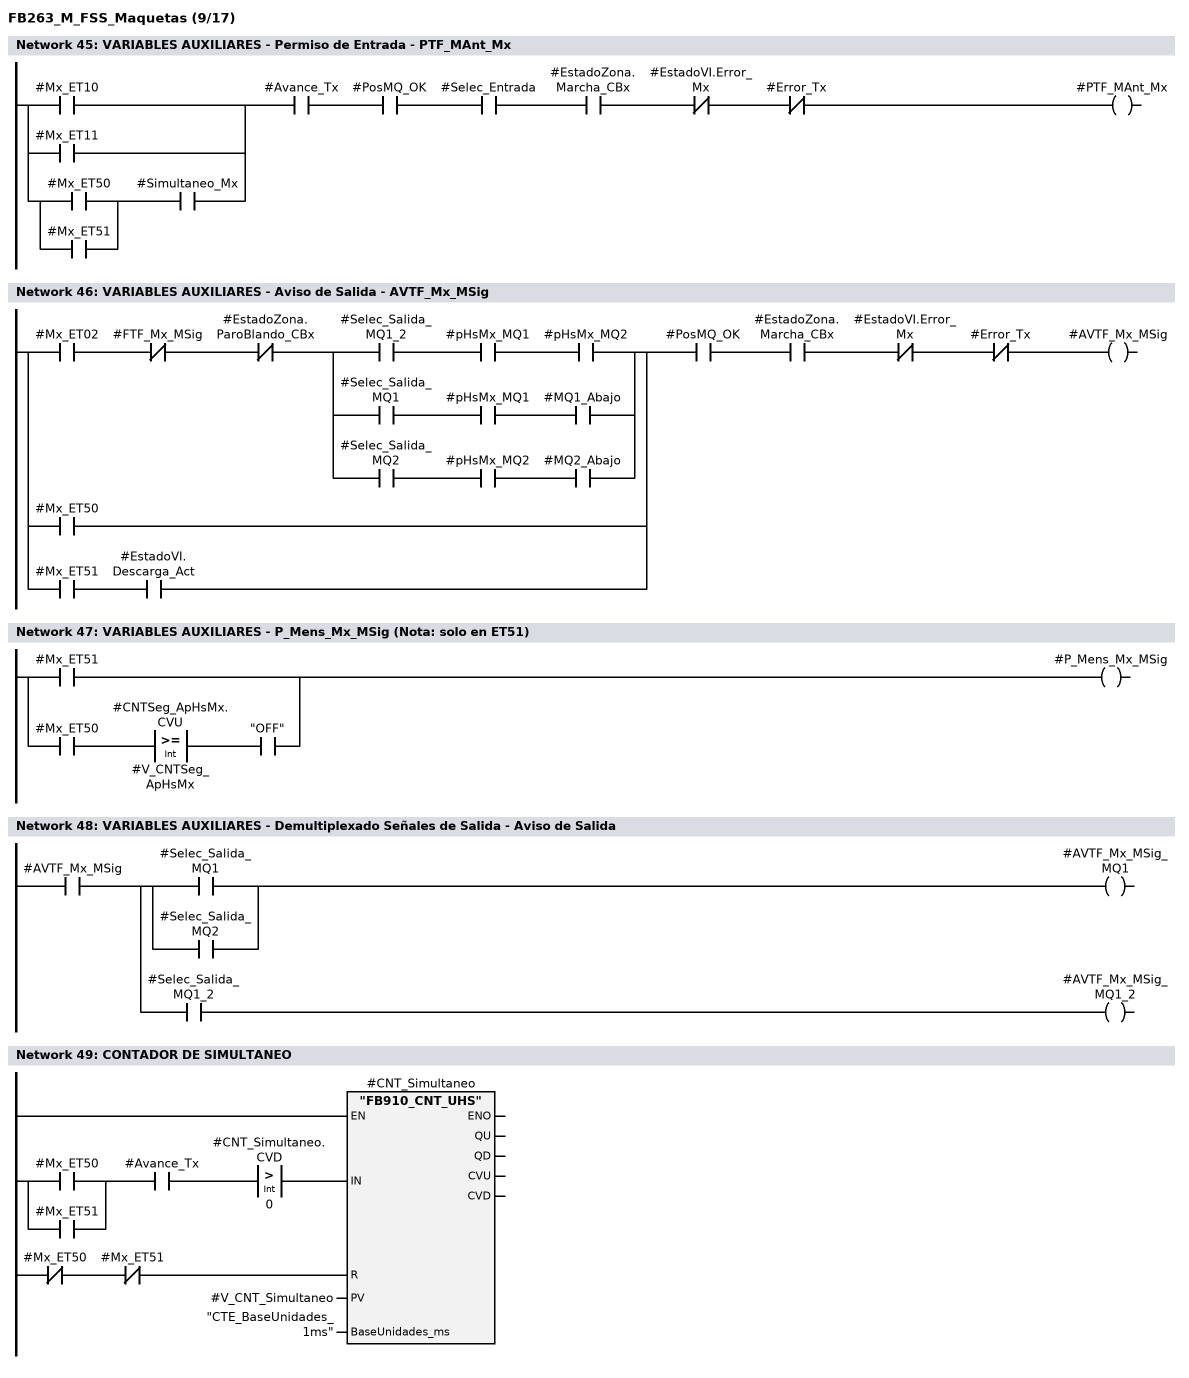
   RUNG wire#powerrail
      Contact( #Mx_ET10 )
      wire#w1
      Contact( #Avance_Tx )
      Contact( #PosMQ_OK )
      Contact( #Selec_Entrada )
      Contact( #EstadoZona.Marcha_CBx )
      I_Contact( #EstadoVI.Error_Mx )
      I_Contact( #Error_Tx )
      Coil( #PTF_MAnt_Mx )
   END_RUNG
   RUNG wire#powerrail
      Contact( #Mx_ET11 )
   END_RUNG wire#w1
   RUNG wire#powerrail
      Contact( #Mx_ET50 )
      wire#w2
      Contact( #Simultaneo_Mx )
   END_RUNG wire#w1
   RUNG wire#powerrail
      Contact( #Mx_ET51 )
   END_RUNG wire#w2
   // the same network as SCL:
   #PTF_MAnt_Mx := (#Mx_ET10 OR #Mx_ET11 OR ((#Mx_ET50 OR #Mx_ET51) AND #Simultaneo_Mx)) AND #Avance_Tx AND #PosMQ_OK AND #Selec_Entrada AND #EstadoZona.Marcha_CBx AND NOT #EstadoVI.Error_Mx AND NOT #Error_Tx;
END_REGION

REGION Network 46: VARIABLES AUXILIARES - Aviso de Salida - AVTF_Mx_MSig
   RUNG wire#powerrail
      Contact( #Mx_ET02 )
      I_Contact( #FTF_Mx_MSig )
      I_Contact( #EstadoZona.ParoBlando_CBx )
      wire#w1
      Contact( #Selec_Salida_MQ1_2 )
      Contact( #pHsMx_MQ1 )
      Contact( #pHsMx_MQ2 )
      wire#w2
      Contact( #PosMQ_OK )
      Contact( #EstadoZona.Marcha_CBx )
      I_Contact( #EstadoVI.Error_Mx )
      I_Contact( #Error_Tx )
      Coil( #AVTF_Mx_MSig )
   END_RUNG
   RUNG wire#w1
      Contact( #Selec_Salida_MQ1 )
      Contact( #pHsMx_MQ1 )
      Contact( #MQ1_Abajo )
   END_RUNG wire#w2
   RUNG wire#w1
      Contact( #Selec_Salida_MQ2 )
      Contact( #pHsMx_MQ2 )
      Contact( #MQ2_Abajo )
   END_RUNG wire#w2
   RUNG wire#powerrail
      Contact( #Mx_ET50 )
   END_RUNG wire#w2
   RUNG wire#powerrail
      Contact( #Mx_ET51 )
      Contact( #EstadoVI.Descarga_Act )
   END_RUNG wire#w2
   // the same network as SCL:
   #AVTF_Mx_MSig := ((#Mx_ET02 AND NOT #FTF_Mx_MSig AND NOT #EstadoZona.ParoBlando_CBx AND ((#Selec_Salida_MQ1_2 AND #pHsMx_MQ1 AND #pHsMx_MQ2) OR (#Selec_Salida_MQ1 AND #pHsMx_MQ1 AND #MQ1_Abajo) OR (#Selec_Salida_MQ2 AND #pHsMx_MQ2 AND #MQ2_Abajo))) OR #Mx_ET50 OR (#Mx_ET51 AND #EstadoVI.Descarga_Act)) AND #PosMQ_OK AND #EstadoZona.Marcha_CBx AND NOT #EstadoVI.Error_Mx AND NOT #Error_Tx;
END_REGION

REGION Network 47: VARIABLES AUXILIARES - P_Mens_Mx_MSig (Nota: solo en ET51)
   RUNG wire#powerrail
      Contact( #Mx_ET51 )
      wire#w1
      Coil( #P_Mens_Mx_MSig )
   END_RUNG
   RUNG wire#powerrail
      Contact( #Mx_ET50 )
      { S7_Templates := "SrcType := Int" } GE_Contact(in1 := #CNTSeg_ApHsMx.CVU, in2 := #V_CNTSeg_ApHsMx)
      Contact( "OFF" )
   END_RUNG wire#w1
   // the same network as SCL:
   #P_Mens_Mx_MSig := #Mx_ET51 OR (#Mx_ET50 AND (#CNTSeg_ApHsMx.CVU >= #V_CNTSeg_ApHsMx) AND "OFF");
END_REGION

REGION Network 48: VARIABLES AUXILIARES - Demultiplexado Señales de Salida - Aviso de Salida
   RUNG wire#powerrail
      Contact( #AVTF_Mx_MSig )
      wire#w1
      Contact( #Selec_Salida_MQ1 )
      wire#w2
      Coil( #AVTF_Mx_MSig_MQ1 )
   END_RUNG
   RUNG wire#w1
      Contact( #Selec_Salida_MQ2 )
   END_RUNG wire#w2
   RUNG wire#w1
      Contact( #Selec_Salida_MQ1_2 )
      Coil( #AVTF_Mx_MSig_MQ1_2 )
   END_RUNG
   // the same network as SCL:
   #AVTF_Mx_MSig_MQ1 := #AVTF_Mx_MSig AND (#Selec_Salida_MQ1 OR #Selec_Salida_MQ2);
   #AVTF_Mx_MSig_MQ1_2 := #AVTF_Mx_MSig AND #Selec_Salida_MQ1_2;
END_REGION

REGION Network 49: CONTADOR DE SIMULTANEO
   RUNG wire#powerrail
      #CNT_Simultaneo(IN := wire#w2, R := wire#w3, PV := #V_CNT_Simultaneo, BaseUnidades_ms := "CTE_BaseUnidades_1ms", QU =>, QD =>, CVU =>, CVD =>)
   END_RUNG
   RUNG wire#powerrail
      Contact( #Mx_ET50 )
      wire#w1
      Contact( #Avance_Tx )
      { S7_Templates := "SrcType := Int" } GT_Contact(in1 := #CNT_Simultaneo.CVD, in2 := 0)
   END_RUNG wire#w2
   RUNG wire#powerrail
      Contact( #Mx_ET51 )
   END_RUNG wire#w1
   RUNG wire#powerrail
      I_Contact( #Mx_ET50 )
      I_Contact( #Mx_ET51 )
   END_RUNG wire#w3
   // the same network as SCL:
   #CNT_Simultaneo(IN := (#Mx_ET50 OR #Mx_ET51) AND #Avance_Tx AND (#CNT_Simultaneo.CVD > 0),   // "FB910_CNT_UHS"
                   R := NOT #Mx_ET50 AND NOT #Mx_ET51,
                   PV := #V_CNT_Simultaneo,
                   BaseUnidades_ms := "CTE_BaseUnidades_1ms");
END_REGION

REGION Network 50: CONTROL DE MOVIMIENTO SIMULTANEO
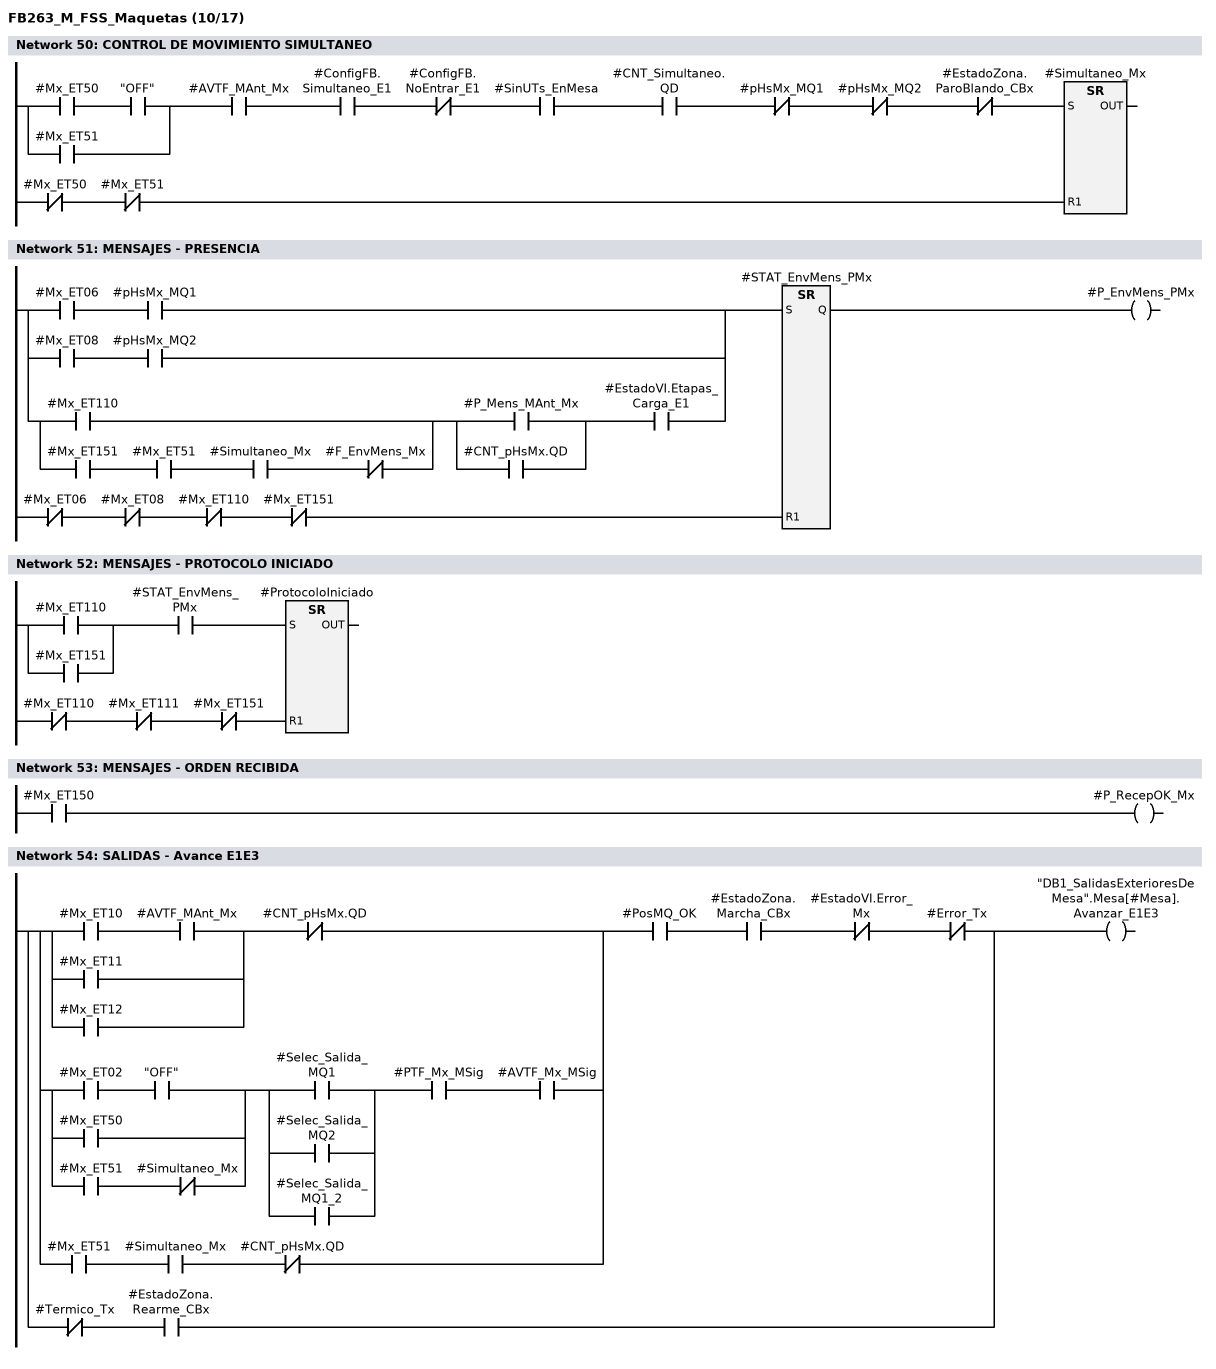
   RUNG wire#powerrail
      Contact( #Mx_ET50 )
      Contact( "OFF" )
      wire#w1
      Contact( #AVTF_MAnt_Mx )
      Contact( #ConfigFB.Simultaneo_E1 )
      I_Contact( #ConfigFB.NoEntrar_E1 )
      Contact( #SinUTs_EnMesa )
      Contact( #CNT_Simultaneo.QD )
      I_Contact( #pHsMx_MQ1 )
      I_Contact( #pHsMx_MQ2 )
      I_Contact( #EstadoZona.ParoBlando_CBx )
      S_SR(operand := #Simultaneo_Mx, r1 := wire#w2)
   END_RUNG
   RUNG wire#powerrail
      Contact( #Mx_ET51 )
   END_RUNG wire#w1
   RUNG wire#powerrail
      I_Contact( #Mx_ET50 )
      I_Contact( #Mx_ET51 )
   END_RUNG wire#w2
   // the same network as SCL:
   IF ((#Mx_ET50 AND "OFF") OR #Mx_ET51) AND #AVTF_MAnt_Mx AND #ConfigFB.Simultaneo_E1 AND NOT #ConfigFB.NoEntrar_E1 AND #SinUTs_EnMesa AND #CNT_Simultaneo.QD AND NOT #pHsMx_MQ1 AND NOT #pHsMx_MQ2 AND NOT #EstadoZona.ParoBlando_CBx THEN
       #Simultaneo_Mx := TRUE;   // SR flip-flop
   END_IF;
   IF NOT #Mx_ET50 AND NOT #Mx_ET51 THEN #Simultaneo_Mx := FALSE; END_IF;
END_REGION

REGION Network 51: MENSAJES - PRESENCIA
   RUNG wire#powerrail
      Contact( #Mx_ET06 )
      Contact( #pHsMx_MQ1 )
      wire#w1
      S_SR(operand := #STAT_EnvMens_PMx, r1 := wire#w4)
      Coil( #P_EnvMens_PMx )
   END_RUNG
   RUNG wire#powerrail
      Contact( #Mx_ET08 )
      Contact( #pHsMx_MQ2 )
   END_RUNG wire#w1
   RUNG wire#powerrail
      Contact( #Mx_ET110 )
      wire#w2
      Contact( #P_Mens_MAnt_Mx )
      wire#w3
      Contact( #EstadoVI.Etapas_Carga_E1 )
   END_RUNG wire#w1
   RUNG wire#powerrail
      Contact( #Mx_ET151 )
      Contact( #Mx_ET51 )
      Contact( #Simultaneo_Mx )
      I_Contact( #F_EnvMens_Mx )
   END_RUNG wire#w2
   RUNG wire#w2
      Contact( #CNT_pHsMx.QD )
   END_RUNG wire#w3
   RUNG wire#powerrail
      I_Contact( #Mx_ET06 )
      I_Contact( #Mx_ET08 )
      I_Contact( #Mx_ET110 )
      I_Contact( #Mx_ET151 )
   END_RUNG wire#w4
   // the same network as SCL:
   IF (#Mx_ET06 AND #pHsMx_MQ1) OR (#Mx_ET08 AND #pHsMx_MQ2) OR ((#Mx_ET110 OR (#Mx_ET151 AND #Mx_ET51 AND #Simultaneo_Mx AND NOT #F_EnvMens_Mx)) AND (#P_Mens_MAnt_Mx OR #CNT_pHsMx.QD) AND #EstadoVI.Etapas_Carga_E1) THEN
       #STAT_EnvMens_PMx := TRUE;   // SR flip-flop
   END_IF;
   IF NOT #Mx_ET06 AND NOT #Mx_ET08 AND NOT #Mx_ET110 AND NOT #Mx_ET151 THEN
       #STAT_EnvMens_PMx := FALSE;
   END_IF;
   #P_EnvMens_PMx := #STAT_EnvMens_PMx;
END_REGION

REGION Network 52: MENSAJES - PROTOCOLO INICIADO
   RUNG wire#powerrail
      Contact( #Mx_ET110 )
      wire#w1
      Contact( #STAT_EnvMens_PMx )
      S_SR(operand := #ProtocoloIniciado, r1 := wire#w2)
   END_RUNG
   RUNG wire#powerrail
      Contact( #Mx_ET151 )
   END_RUNG wire#w1
   RUNG wire#powerrail
      I_Contact( #Mx_ET110 )
      I_Contact( #Mx_ET111 )
      I_Contact( #Mx_ET151 )
   END_RUNG wire#w2
   // the same network as SCL:
   IF (#Mx_ET110 OR #Mx_ET151) AND #STAT_EnvMens_PMx THEN
       #ProtocoloIniciado := TRUE;   // SR flip-flop
   END_IF;
   IF NOT #Mx_ET110 AND NOT #Mx_ET111 AND NOT #Mx_ET151 THEN #ProtocoloIniciado := FALSE; END_IF;
END_REGION

REGION Network 53: MENSAJES - ORDEN RECIBIDA
   RUNG wire#powerrail
      Contact( #Mx_ET150 )
      Coil( #P_RecepOK_Mx )
   END_RUNG
   // the same network as SCL:
   #P_RecepOK_Mx := #Mx_ET150;
END_REGION

REGION Network 54: SALIDAS - Avance E1E3
   RUNG wire#powerrail
      Contact( #Mx_ET10 )
      Contact( #AVTF_MAnt_Mx )
      wire#w1
      I_Contact( #CNT_pHsMx.QD )
      wire#w2
      Contact( #PosMQ_OK )
      Contact( #EstadoZona.Marcha_CBx )
      I_Contact( #EstadoVI.Error_Mx )
      I_Contact( #Error_Tx )
      wire#w5
      Coil( "DB1_SalidasExterioresDeMesa".Mesa[#Mesa].Avanzar_E1E3 )
   END_RUNG
   RUNG wire#powerrail
      Contact( #Mx_ET11 )
   END_RUNG wire#w1
   RUNG wire#powerrail
      Contact( #Mx_ET12 )
   END_RUNG wire#w1
   RUNG wire#powerrail
      Contact( #Mx_ET02 )
      Contact( "OFF" )
      wire#w3
      Contact( #Selec_Salida_MQ1 )
      wire#w4
      Contact( #PTF_Mx_MSig )
      Contact( #AVTF_Mx_MSig )
   END_RUNG wire#w2
   RUNG wire#powerrail
      Contact( #Mx_ET50 )
   END_RUNG wire#w3
   RUNG wire#powerrail
      Contact( #Mx_ET51 )
      I_Contact( #Simultaneo_Mx )
   END_RUNG wire#w3
   RUNG wire#w3
      Contact( #Selec_Salida_MQ2 )
   END_RUNG wire#w4
   RUNG wire#w3
      Contact( #Selec_Salida_MQ1_2 )
   END_RUNG wire#w4
   RUNG wire#powerrail
      Contact( #Mx_ET51 )
      Contact( #Simultaneo_Mx )
      I_Contact( #CNT_pHsMx.QD )
   END_RUNG wire#w2
   RUNG wire#powerrail
      I_Contact( #Termico_Tx )
      Contact( #EstadoZona.Rearme_CBx )
   END_RUNG wire#w5
   // the same network as SCL:
   "DB1_SalidasExterioresDeMesa".Mesa[#Mesa].Avanzar_E1E3 := (((((#Mx_ET10 AND #AVTF_MAnt_Mx) OR #Mx_ET11 OR #Mx_ET12) AND NOT #CNT_pHsMx.QD) OR (((#Mx_ET02 AND "OFF") OR #Mx_ET50 OR (#Mx_ET51 AND NOT #Simultaneo_Mx)) AND (#Selec_Salida_MQ1 OR #Selec_Salida_MQ2 OR #Selec_Salida_MQ1_2) AND #PTF_Mx_MSig AND #AVTF_Mx_MSig) OR (#Mx_ET51 AND #Simultaneo_Mx AND NOT #CNT_pHsMx.QD)) AND #PosMQ_OK AND #EstadoZona.Marcha_CBx AND NOT #EstadoVI.Error_Mx AND NOT #Error_Tx) OR (NOT #Termico_Tx AND #EstadoZona.Rearme_CBx);
END_REGION

REGION Network 55: SALIDAS - Subir Tope (TP1)
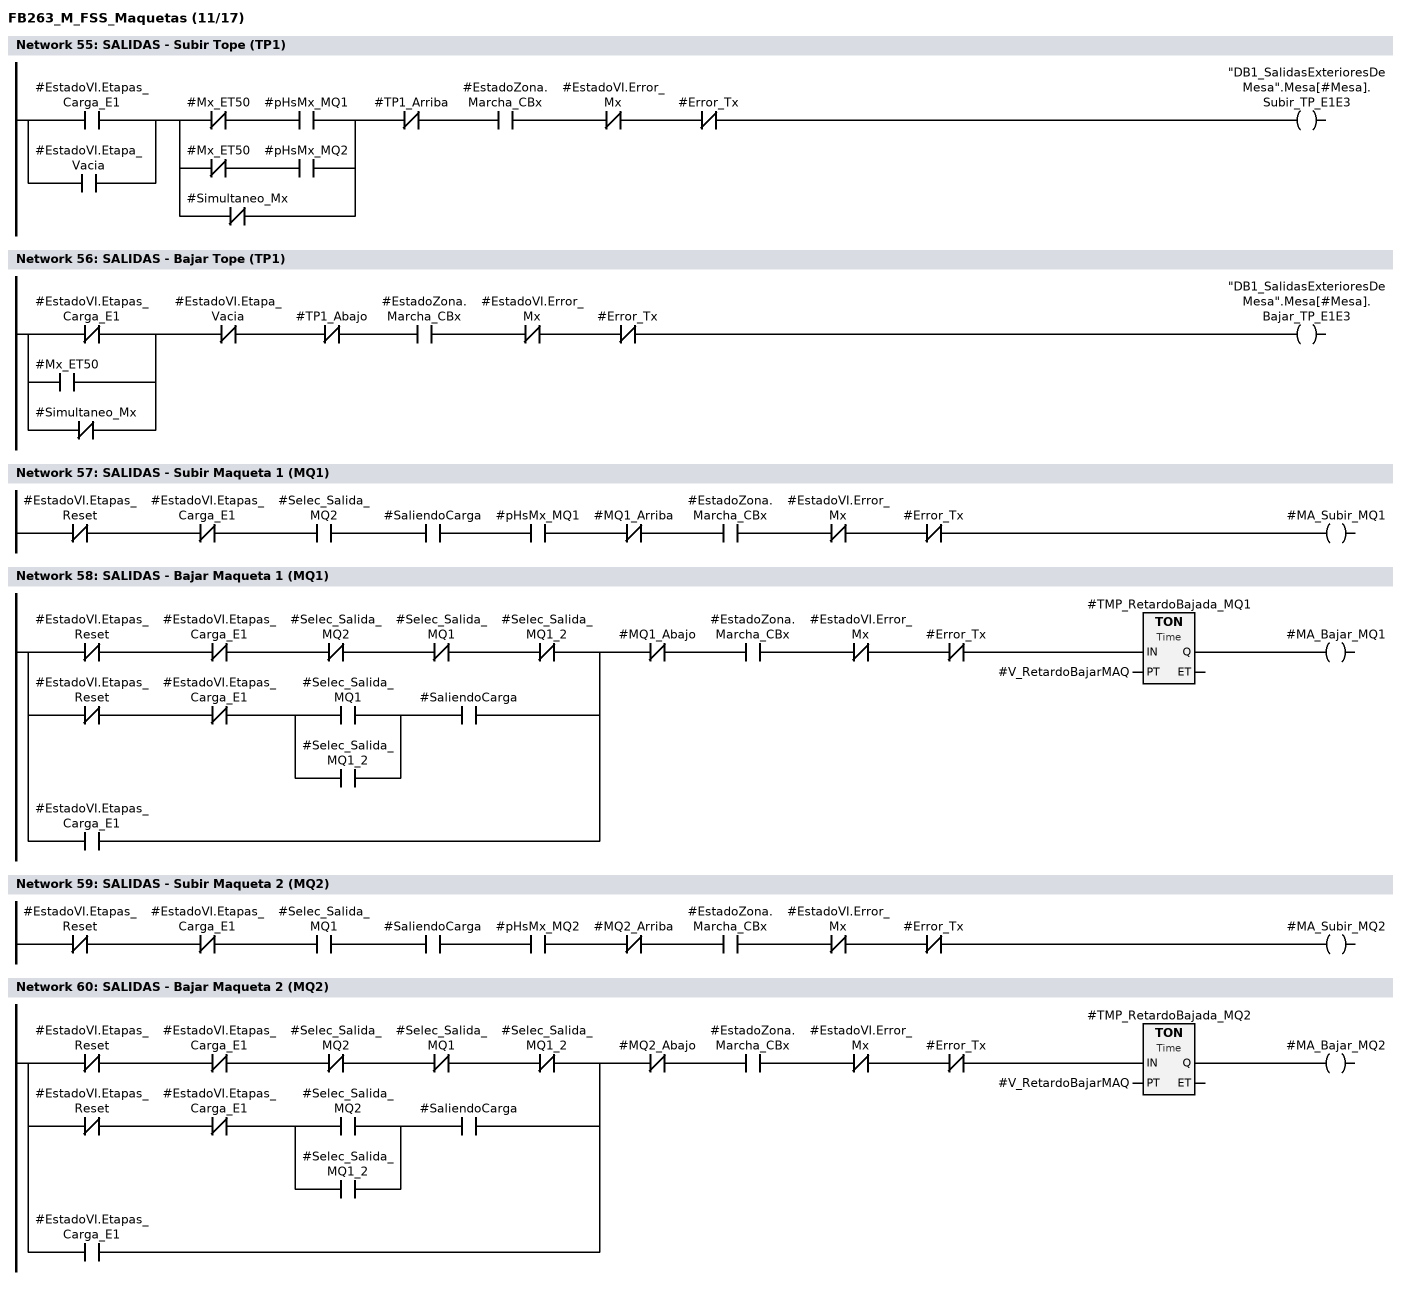
   RUNG wire#powerrail
      Contact( #EstadoVI.Etapas_Carga_E1 )
      wire#w1
      I_Contact( #Mx_ET50 )
      Contact( #pHsMx_MQ1 )
      wire#w2
      I_Contact( #TP1_Arriba )
      Contact( #EstadoZona.Marcha_CBx )
      I_Contact( #EstadoVI.Error_Mx )
      I_Contact( #Error_Tx )
      Coil( "DB1_SalidasExterioresDeMesa".Mesa[#Mesa].Subir_TP_E1E3 )
   END_RUNG
   RUNG wire#powerrail
      Contact( #EstadoVI.Etapa_Vacia )
   END_RUNG wire#w1
   RUNG wire#w1
      I_Contact( #Mx_ET50 )
      Contact( #pHsMx_MQ2 )
   END_RUNG wire#w2
   RUNG wire#w1
      I_Contact( #Simultaneo_Mx )
   END_RUNG wire#w2
   // the same network as SCL:
   "DB1_SalidasExterioresDeMesa".Mesa[#Mesa].Subir_TP_E1E3 := (#EstadoVI.Etapas_Carga_E1 OR #EstadoVI.Etapa_Vacia) AND ((NOT #Mx_ET50 AND #pHsMx_MQ1) OR (NOT #Mx_ET50 AND #pHsMx_MQ2) OR NOT #Simultaneo_Mx) AND NOT #TP1_Arriba AND #EstadoZona.Marcha_CBx AND NOT #EstadoVI.Error_Mx AND NOT #Error_Tx;
END_REGION

REGION Network 56: SALIDAS - Bajar Tope (TP1)
   RUNG wire#powerrail
      I_Contact( #EstadoVI.Etapas_Carga_E1 )
      wire#w1
      I_Contact( #EstadoVI.Etapa_Vacia )
      I_Contact( #TP1_Abajo )
      Contact( #EstadoZona.Marcha_CBx )
      I_Contact( #EstadoVI.Error_Mx )
      I_Contact( #Error_Tx )
      Coil( "DB1_SalidasExterioresDeMesa".Mesa[#Mesa].Bajar_TP_E1E3 )
   END_RUNG
   RUNG wire#powerrail
      Contact( #Mx_ET50 )
   END_RUNG wire#w1
   RUNG wire#powerrail
      I_Contact( #Simultaneo_Mx )
   END_RUNG wire#w1
   // the same network as SCL:
   "DB1_SalidasExterioresDeMesa".Mesa[#Mesa].Bajar_TP_E1E3 := (NOT #EstadoVI.Etapas_Carga_E1 OR #Mx_ET50 OR NOT #Simultaneo_Mx) AND NOT #EstadoVI.Etapa_Vacia AND NOT #TP1_Abajo AND #EstadoZona.Marcha_CBx AND NOT #EstadoVI.Error_Mx AND NOT #Error_Tx;
END_REGION

REGION Network 57: SALIDAS - Subir Maqueta 1 (MQ1)
   RUNG wire#powerrail
      I_Contact( #EstadoVI.Etapas_Reset )
      I_Contact( #EstadoVI.Etapas_Carga_E1 )
      Contact( #Selec_Salida_MQ2 )
      Contact( #SaliendoCarga )
      Contact( #pHsMx_MQ1 )
      I_Contact( #MQ1_Arriba )
      Contact( #EstadoZona.Marcha_CBx )
      I_Contact( #EstadoVI.Error_Mx )
      I_Contact( #Error_Tx )
      Coil( #MA_Subir_MQ1 )
   END_RUNG
   // the same network as SCL:
   #MA_Subir_MQ1 := NOT #EstadoVI.Etapas_Reset AND NOT #EstadoVI.Etapas_Carga_E1 AND #Selec_Salida_MQ2 AND #SaliendoCarga AND #pHsMx_MQ1 AND NOT #MQ1_Arriba AND #EstadoZona.Marcha_CBx AND NOT #EstadoVI.Error_Mx AND NOT #Error_Tx;
END_REGION

REGION Network 58: SALIDAS - Bajar Maqueta 1 (MQ1)
   RUNG wire#powerrail
      I_Contact( #EstadoVI.Etapas_Reset )
      I_Contact( #EstadoVI.Etapas_Carga_E1 )
      I_Contact( #Selec_Salida_MQ2 )
      I_Contact( #Selec_Salida_MQ1 )
      I_Contact( #Selec_Salida_MQ1_2 )
      wire#w1
      I_Contact( #MQ1_Abajo )
      Contact( #EstadoZona.Marcha_CBx )
      I_Contact( #EstadoVI.Error_Mx )
      I_Contact( #Error_Tx )
      { S7_Templates := "time_type := Time" } #TMP_RetardoBajada_MQ1.TON(pt := #V_RetardoBajarMAQ, et =>)
      Coil( #MA_Bajar_MQ1 )
   END_RUNG
   RUNG wire#powerrail
      I_Contact( #EstadoVI.Etapas_Reset )
      I_Contact( #EstadoVI.Etapas_Carga_E1 )
      wire#w2
      Contact( #Selec_Salida_MQ1 )
      wire#w3
      Contact( #SaliendoCarga )
   END_RUNG wire#w1
   RUNG wire#w2
      Contact( #Selec_Salida_MQ1_2 )
   END_RUNG wire#w3
   RUNG wire#powerrail
      Contact( #EstadoVI.Etapas_Carga_E1 )
   END_RUNG wire#w1
   // the same network as SCL:
   #TMP_RetardoBajada_MQ1(IN := ((NOT #EstadoVI.Etapas_Reset AND NOT #EstadoVI.Etapas_Carga_E1 AND NOT #Selec_Salida_MQ2 AND NOT #Selec_Salida_MQ1 AND NOT #Selec_Salida_MQ1_2) OR (NOT #EstadoVI.Etapas_Reset AND NOT #EstadoVI.Etapas_Carga_E1 AND (#Selec_Salida_MQ1 OR #Selec_Salida_MQ1_2) AND #SaliendoCarga) OR #EstadoVI.Etapas_Carga_E1) AND NOT #MQ1_Abajo AND #EstadoZona.Marcha_CBx AND NOT #EstadoVI.Error_Mx AND NOT #Error_Tx,   // TON
                          PT := #V_RetardoBajarMAQ);
   #MA_Bajar_MQ1 := #TMP_RetardoBajada_MQ1.Q;
END_REGION

REGION Network 59: SALIDAS - Subir Maqueta 2 (MQ2)
   RUNG wire#powerrail
      I_Contact( #EstadoVI.Etapas_Reset )
      I_Contact( #EstadoVI.Etapas_Carga_E1 )
      Contact( #Selec_Salida_MQ1 )
      Contact( #SaliendoCarga )
      Contact( #pHsMx_MQ2 )
      I_Contact( #MQ2_Arriba )
      Contact( #EstadoZona.Marcha_CBx )
      I_Contact( #EstadoVI.Error_Mx )
      I_Contact( #Error_Tx )
      Coil( #MA_Subir_MQ2 )
   END_RUNG
   // the same network as SCL:
   #MA_Subir_MQ2 := NOT #EstadoVI.Etapas_Reset AND NOT #EstadoVI.Etapas_Carga_E1 AND #Selec_Salida_MQ1 AND #SaliendoCarga AND #pHsMx_MQ2 AND NOT #MQ2_Arriba AND #EstadoZona.Marcha_CBx AND NOT #EstadoVI.Error_Mx AND NOT #Error_Tx;
END_REGION

REGION Network 60: SALIDAS - Bajar Maqueta 2 (MQ2)
   RUNG wire#powerrail
      I_Contact( #EstadoVI.Etapas_Reset )
      I_Contact( #EstadoVI.Etapas_Carga_E1 )
      I_Contact( #Selec_Salida_MQ2 )
      I_Contact( #Selec_Salida_MQ1 )
      I_Contact( #Selec_Salida_MQ1_2 )
      wire#w1
      I_Contact( #MQ2_Abajo )
      Contact( #EstadoZona.Marcha_CBx )
      I_Contact( #EstadoVI.Error_Mx )
      I_Contact( #Error_Tx )
      { S7_Templates := "time_type := Time" } #TMP_RetardoBajada_MQ2.TON(pt := #V_RetardoBajarMAQ, et =>)
      Coil( #MA_Bajar_MQ2 )
   END_RUNG
   RUNG wire#powerrail
      I_Contact( #EstadoVI.Etapas_Reset )
      I_Contact( #EstadoVI.Etapas_Carga_E1 )
      wire#w2
      Contact( #Selec_Salida_MQ2 )
      wire#w3
      Contact( #SaliendoCarga )
   END_RUNG wire#w1
   RUNG wire#w2
      Contact( #Selec_Salida_MQ1_2 )
   END_RUNG wire#w3
   RUNG wire#powerrail
      Contact( #EstadoVI.Etapas_Carga_E1 )
   END_RUNG wire#w1
   // the same network as SCL:
   #TMP_RetardoBajada_MQ2(IN := ((NOT #EstadoVI.Etapas_Reset AND NOT #EstadoVI.Etapas_Carga_E1 AND NOT #Selec_Salida_MQ2 AND NOT #Selec_Salida_MQ1 AND NOT #Selec_Salida_MQ1_2) OR (NOT #EstadoVI.Etapas_Reset AND NOT #EstadoVI.Etapas_Carga_E1 AND (#Selec_Salida_MQ2 OR #Selec_Salida_MQ1_2) AND #SaliendoCarga) OR #EstadoVI.Etapas_Carga_E1) AND NOT #MQ2_Abajo AND #EstadoZona.Marcha_CBx AND NOT #EstadoVI.Error_Mx AND NOT #Error_Tx,   // TON
                          PT := #V_RetardoBajarMAQ);
   #MA_Bajar_MQ2 := #TMP_RetardoBajada_MQ2.Q;
END_REGION

REGION Network 61: TMP - Espera En Tension
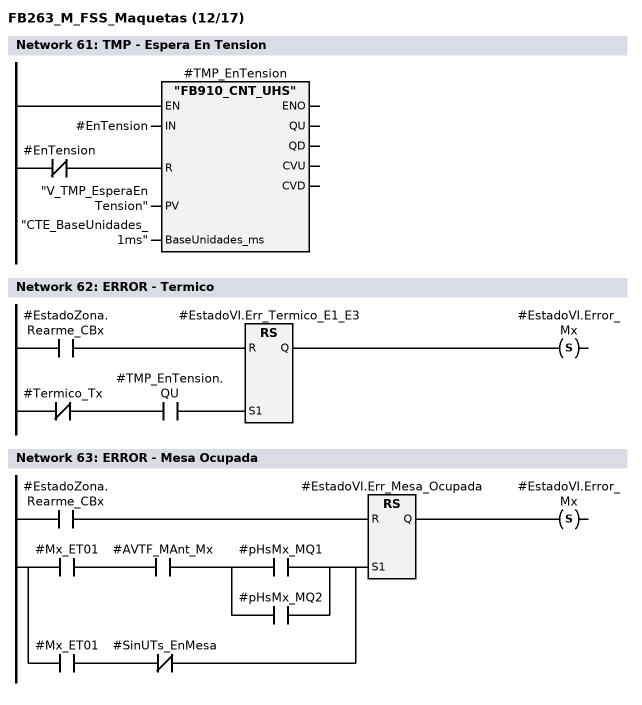
   RUNG wire#powerrail
      #TMP_EnTension(R := wire#w1, IN := #EnTension, PV := "V_TMP_EsperaEnTension", BaseUnidades_ms := "CTE_BaseUnidades_1ms", QU =>, QD =>, CVU =>, CVD =>)
   END_RUNG
   RUNG wire#powerrail
      I_Contact( #EnTension )
   END_RUNG wire#w1
   // the same network as SCL:
   #TMP_EnTension(IN := #EnTension,   // "FB910_CNT_UHS"
                  R := NOT #EnTension,
                  PV := "V_TMP_EsperaEnTension",
                  BaseUnidades_ms := "CTE_BaseUnidades_1ms");
END_REGION

REGION Network 62: ERROR - Termico
   RUNG wire#powerrail
      Contact( #EstadoZona.Rearme_CBx )
      S_RS(operand := #EstadoVI.Err_Termico_E1_E3, s1 := wire#w1)
      S_Coil( #EstadoVI.Error_Mx )
   END_RUNG
   RUNG wire#powerrail
      I_Contact( #Termico_Tx )
      Contact( #TMP_EnTension.QU )
   END_RUNG wire#w1
   // the same network as SCL:
   IF #EstadoZona.Rearme_CBx THEN
       #EstadoVI.Err_Termico_E1_E3 := FALSE;   // RS flip-flop
   END_IF;
   IF NOT #Termico_Tx AND #TMP_EnTension.QU THEN #EstadoVI.Err_Termico_E1_E3 := TRUE; END_IF;
   IF #EstadoVI.Err_Termico_E1_E3 THEN #EstadoVI.Error_Mx := TRUE; END_IF;
END_REGION

REGION Network 63: ERROR - Mesa Ocupada
   RUNG wire#powerrail
      Contact( #EstadoZona.Rearme_CBx )
      S_RS(operand := #EstadoVI.Err_Mesa_Ocupada, s1 := wire#w2)
      S_Coil( #EstadoVI.Error_Mx )
   END_RUNG
   RUNG wire#powerrail
      Contact( #Mx_ET01 )
      Contact( #AVTF_MAnt_Mx )
      wire#w1
      Contact( #pHsMx_MQ1 )
   END_RUNG wire#w2
   RUNG wire#w1
      Contact( #pHsMx_MQ2 )
   END_RUNG wire#w2
   RUNG wire#powerrail
      Contact( #Mx_ET01 )
      I_Contact( #SinUTs_EnMesa )
   END_RUNG wire#w2
   // the same network as SCL:
   IF #EstadoZona.Rearme_CBx THEN
       #EstadoVI.Err_Mesa_Ocupada := FALSE;   // RS flip-flop
   END_IF;
   IF (#Mx_ET01 AND #AVTF_MAnt_Mx AND (#pHsMx_MQ1 OR #pHsMx_MQ2)) OR (#Mx_ET01 AND NOT #SinUTs_EnMesa) THEN
       #EstadoVI.Err_Mesa_Ocupada := TRUE;
   END_IF;
   IF #EstadoVI.Err_Mesa_Ocupada THEN #EstadoVI.Error_Mx := TRUE; END_IF;
END_REGION

REGION Network 64: CNT - ERROR - Arrastre
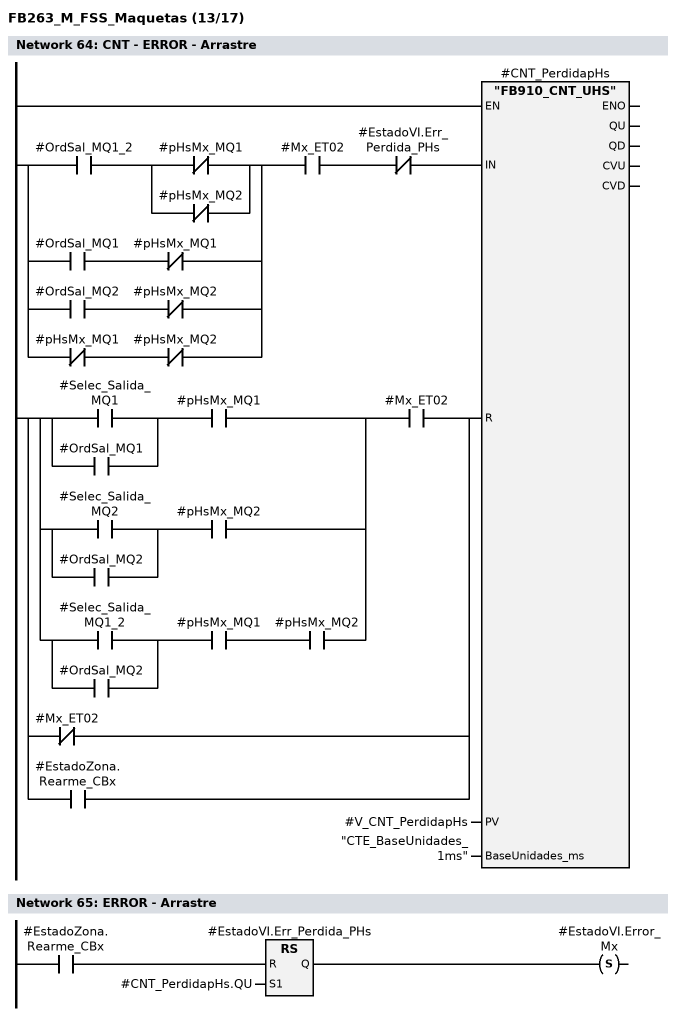
   RUNG wire#powerrail
      #CNT_PerdidapHs(IN := wire#w3, R := wire#w8, PV := #V_CNT_PerdidapHs, BaseUnidades_ms := "CTE_BaseUnidades_1ms", QU =>, QD =>, CVU =>, CVD =>)
   END_RUNG
   RUNG wire#powerrail
      Contact( #OrdSal_MQ1_2 )
      wire#w1
      I_Contact( #pHsMx_MQ1 )
      wire#w2
      Contact( #Mx_ET02 )
      I_Contact( #EstadoVI.Err_Perdida_PHs )
   END_RUNG wire#w3
   RUNG wire#w1
      I_Contact( #pHsMx_MQ2 )
   END_RUNG wire#w2
   RUNG wire#powerrail
      Contact( #OrdSal_MQ1 )
      I_Contact( #pHsMx_MQ1 )
   END_RUNG wire#w2
   RUNG wire#powerrail
      Contact( #OrdSal_MQ2 )
      I_Contact( #pHsMx_MQ2 )
   END_RUNG wire#w2
   RUNG wire#powerrail
      I_Contact( #pHsMx_MQ1 )
      I_Contact( #pHsMx_MQ2 )
   END_RUNG wire#w2
   RUNG wire#powerrail
      Contact( #Selec_Salida_MQ1 )
      wire#w4
      Contact( #pHsMx_MQ1 )
      wire#w5
      Contact( #Mx_ET02 )
   END_RUNG wire#w8
   RUNG wire#powerrail
      Contact( #OrdSal_MQ1 )
   END_RUNG wire#w4
   RUNG wire#powerrail
      Contact( #Selec_Salida_MQ2 )
      wire#w6
      Contact( #pHsMx_MQ2 )
   END_RUNG wire#w5
   RUNG wire#powerrail
      Contact( #OrdSal_MQ2 )
   END_RUNG wire#w6
   RUNG wire#powerrail
      Contact( #Selec_Salida_MQ1_2 )
      wire#w7
      Contact( #pHsMx_MQ1 )
      Contact( #pHsMx_MQ2 )
   END_RUNG wire#w5
   RUNG wire#powerrail
      Contact( #OrdSal_MQ2 )
   END_RUNG wire#w7
   RUNG wire#powerrail
      I_Contact( #Mx_ET02 )
   END_RUNG wire#w8
   RUNG wire#powerrail
      Contact( #EstadoZona.Rearme_CBx )
   END_RUNG wire#w8
   // the same network as SCL:
   #CNT_PerdidapHs(IN := ((#OrdSal_MQ1_2 AND (NOT #pHsMx_MQ1 OR NOT #pHsMx_MQ2)) OR (#OrdSal_MQ1 AND NOT #pHsMx_MQ1) OR (#OrdSal_MQ2 AND NOT #pHsMx_MQ2) OR (NOT #pHsMx_MQ1 AND NOT #pHsMx_MQ2)) AND #Mx_ET02 AND NOT #EstadoVI.Err_Perdida_PHs,   // "FB910_CNT_UHS"
                   R := ((((#Selec_Salida_MQ1 OR #OrdSal_MQ1) AND #pHsMx_MQ1) OR ((#Selec_Salida_MQ2 OR #OrdSal_MQ2) AND #pHsMx_MQ2) OR ((#Selec_Salida_MQ1_2 OR #OrdSal_MQ2) AND #pHsMx_MQ1 AND #pHsMx_MQ2)) AND #Mx_ET02) OR NOT #Mx_ET02 OR #EstadoZona.Rearme_CBx,
                   PV := #V_CNT_PerdidapHs,
                   BaseUnidades_ms := "CTE_BaseUnidades_1ms");
END_REGION

REGION Network 65: ERROR - Arrastre
   RUNG wire#powerrail
      Contact( #EstadoZona.Rearme_CBx )
      S_RS(operand := #EstadoVI.Err_Perdida_PHs, s1 := #CNT_PerdidapHs.QU)
      S_Coil( #EstadoVI.Error_Mx )
   END_RUNG
   // the same network as SCL:
   IF #EstadoZona.Rearme_CBx THEN
       #EstadoVI.Err_Perdida_PHs := FALSE;   // RS flip-flop
   END_IF;
   IF #CNT_PerdidapHs.QU THEN #EstadoVI.Err_Perdida_PHs := TRUE; END_IF;
   IF #EstadoVI.Err_Perdida_PHs THEN #EstadoVI.Error_Mx := TRUE; END_IF;
END_REGION

REGION Network 66: ERROR - Descarga por S3
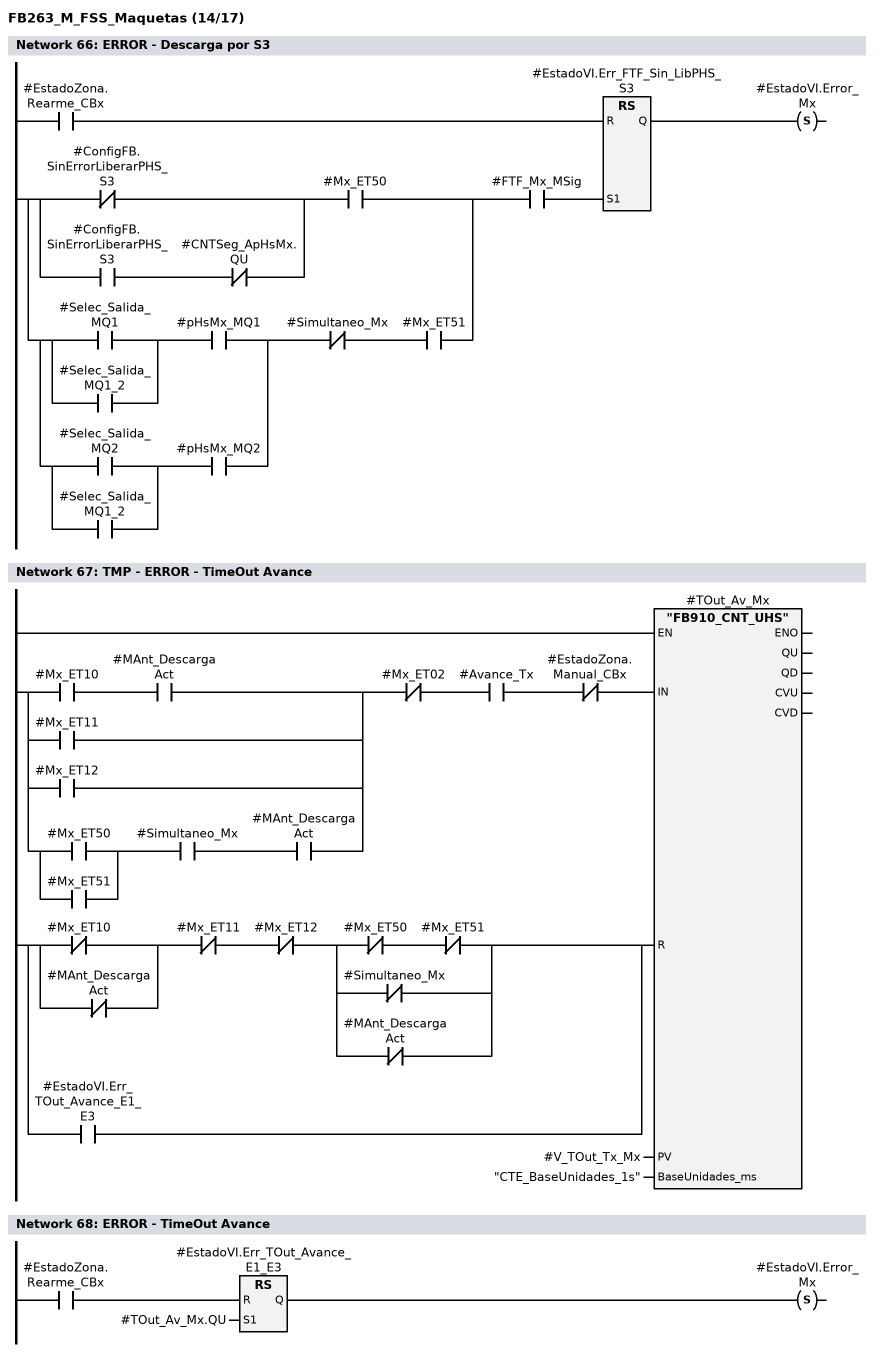
   RUNG wire#powerrail
      Contact( #EstadoZona.Rearme_CBx )
      S_RS(operand := #EstadoVI.Err_FTF_Sin_LibPHS_S3, s1 := wire#w6)
      S_Coil( #EstadoVI.Error_Mx )
   END_RUNG
   RUNG wire#powerrail
      I_Contact( #ConfigFB.SinErrorLiberarPHS_S3 )
      wire#w1
      Contact( #Mx_ET50 )
      wire#w2
      Contact( #FTF_Mx_MSig )
   END_RUNG wire#w6
   RUNG wire#powerrail
      Contact( #ConfigFB.SinErrorLiberarPHS_S3 )
      I_Contact( #CNTSeg_ApHsMx.QU )
   END_RUNG wire#w1
   RUNG wire#powerrail
      Contact( #Selec_Salida_MQ1 )
      wire#w3
      Contact( #pHsMx_MQ1 )
      wire#w4
      I_Contact( #Simultaneo_Mx )
      Contact( #Mx_ET51 )
   END_RUNG wire#w2
   RUNG wire#powerrail
      Contact( #Selec_Salida_MQ1_2 )
   END_RUNG wire#w3
   RUNG wire#powerrail
      Contact( #Selec_Salida_MQ2 )
      wire#w5
      Contact( #pHsMx_MQ2 )
   END_RUNG wire#w4
   RUNG wire#powerrail
      Contact( #Selec_Salida_MQ1_2 )
   END_RUNG wire#w5
   // the same network as SCL:
   IF #EstadoZona.Rearme_CBx THEN
       #EstadoVI.Err_FTF_Sin_LibPHS_S3 := FALSE;   // RS flip-flop
   END_IF;
   IF (((NOT #ConfigFB.SinErrorLiberarPHS_S3 OR (#ConfigFB.SinErrorLiberarPHS_S3 AND NOT #CNTSeg_ApHsMx.QU)) AND #Mx_ET50) OR ((((#Selec_Salida_MQ1 OR #Selec_Salida_MQ1_2) AND #pHsMx_MQ1) OR ((#Selec_Salida_MQ2 OR #Selec_Salida_MQ1_2) AND #pHsMx_MQ2)) AND NOT #Simultaneo_Mx AND #Mx_ET51)) AND #FTF_Mx_MSig THEN
       #EstadoVI.Err_FTF_Sin_LibPHS_S3 := TRUE;
   END_IF;
   IF #EstadoVI.Err_FTF_Sin_LibPHS_S3 THEN #EstadoVI.Error_Mx := TRUE; END_IF;
END_REGION

REGION Network 67: TMP - ERROR - TimeOut Avance
   RUNG wire#powerrail
      #TOut_Av_Mx(IN := wire#w3, R := wire#w6, PV := #V_TOut_Tx_Mx, BaseUnidades_ms := "CTE_BaseUnidades_1s", QU =>, QD =>, CVU =>, CVD =>)
   END_RUNG
   RUNG wire#powerrail
      Contact( #Mx_ET10 )
      Contact( #MAnt_DescargaAct )
      wire#w1
      I_Contact( #Mx_ET02 )
      Contact( #Avance_Tx )
      I_Contact( #EstadoZona.Manual_CBx )
   END_RUNG wire#w3
   RUNG wire#powerrail
      Contact( #Mx_ET11 )
   END_RUNG wire#w1
   RUNG wire#powerrail
      Contact( #Mx_ET12 )
   END_RUNG wire#w1
   RUNG wire#powerrail
      Contact( #Mx_ET50 )
      wire#w2
      Contact( #Simultaneo_Mx )
      Contact( #MAnt_DescargaAct )
   END_RUNG wire#w1
   RUNG wire#powerrail
      Contact( #Mx_ET51 )
   END_RUNG wire#w2
   RUNG wire#powerrail
      I_Contact( #Mx_ET10 )
      wire#w4
      I_Contact( #Mx_ET11 )
      I_Contact( #Mx_ET12 )
      wire#w5
      I_Contact( #Mx_ET50 )
      I_Contact( #Mx_ET51 )
   END_RUNG wire#w6
   RUNG wire#powerrail
      I_Contact( #MAnt_DescargaAct )
   END_RUNG wire#w4
   RUNG wire#w5
      I_Contact( #Simultaneo_Mx )
   END_RUNG wire#w6
   RUNG wire#w5
      I_Contact( #MAnt_DescargaAct )
   END_RUNG wire#w6
   RUNG wire#powerrail
      Contact( #EstadoVI.Err_TOut_Avance_E1_E3 )
   END_RUNG wire#w6
   // the same network as SCL:
   #TOut_Av_Mx(IN := ((#Mx_ET10 AND #MAnt_DescargaAct) OR #Mx_ET11 OR #Mx_ET12 OR ((#Mx_ET50 OR #Mx_ET51) AND #Simultaneo_Mx AND #MAnt_DescargaAct)) AND NOT #Mx_ET02 AND #Avance_Tx AND NOT #EstadoZona.Manual_CBx,   // "FB910_CNT_UHS"
               R := ((NOT #Mx_ET10 OR NOT #MAnt_DescargaAct) AND NOT #Mx_ET11 AND NOT #Mx_ET12 AND ((NOT #Mx_ET50 AND NOT #Mx_ET51) OR NOT #Simultaneo_Mx OR NOT #MAnt_DescargaAct)) OR #EstadoVI.Err_TOut_Avance_E1_E3,
               PV := #V_TOut_Tx_Mx,
               BaseUnidades_ms := "CTE_BaseUnidades_1s");
END_REGION

REGION Network 68: ERROR - TimeOut Avance
   RUNG wire#powerrail
      Contact( #EstadoZona.Rearme_CBx )
      S_RS(operand := #EstadoVI.Err_TOut_Avance_E1_E3, s1 := #TOut_Av_Mx.QU)
      S_Coil( #EstadoVI.Error_Mx )
   END_RUNG
   // the same network as SCL:
   IF #EstadoZona.Rearme_CBx THEN
       #EstadoVI.Err_TOut_Avance_E1_E3 := FALSE;   // RS flip-flop
   END_IF;
   IF #TOut_Av_Mx.QU THEN #EstadoVI.Err_TOut_Avance_E1_E3 := TRUE; END_IF;
   IF #EstadoVI.Err_TOut_Avance_E1_E3 THEN #EstadoVI.Error_Mx := TRUE; END_IF;
END_REGION

REGION Network 69: TMP - ERROR - TimeOut Subir TP
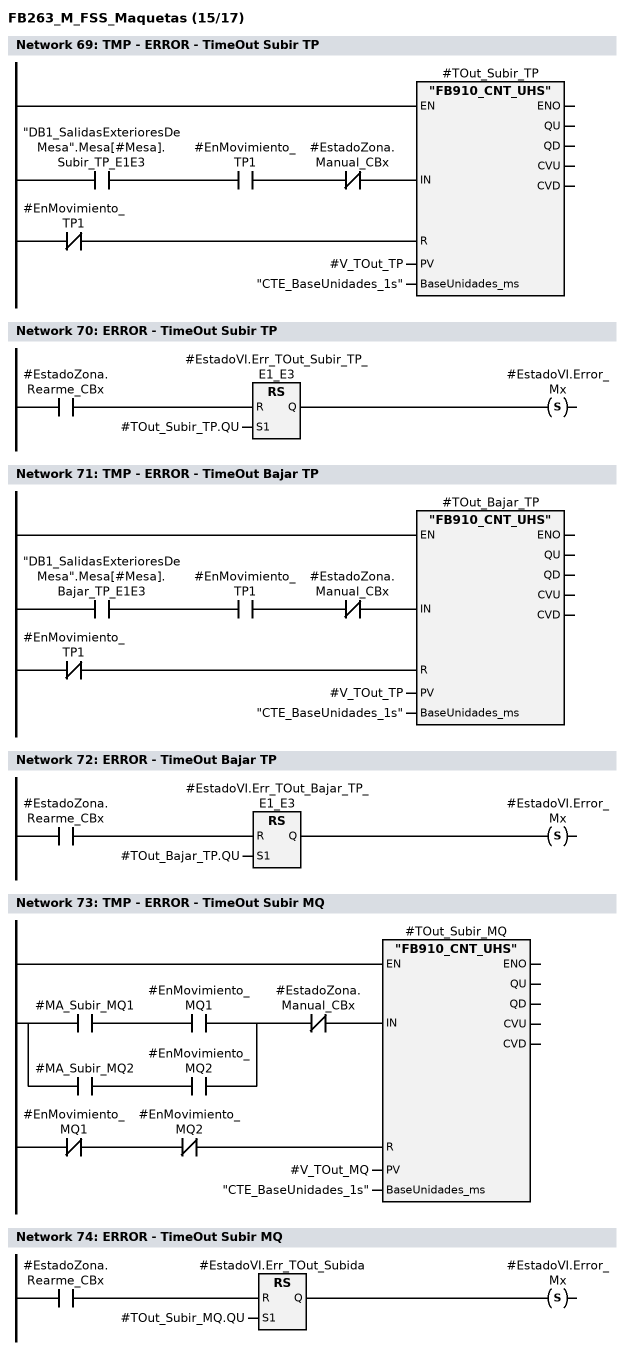
   RUNG wire#powerrail
      #TOut_Subir_TP(IN := wire#w1, R := wire#w2, PV := #V_TOut_TP, BaseUnidades_ms := "CTE_BaseUnidades_1s", QU =>, QD =>, CVU =>, CVD =>)
   END_RUNG
   RUNG wire#powerrail
      Contact( "DB1_SalidasExterioresDeMesa".Mesa[#Mesa].Subir_TP_E1E3 )
      Contact( #EnMovimiento_TP1 )
      I_Contact( #EstadoZona.Manual_CBx )
   END_RUNG wire#w1
   RUNG wire#powerrail
      I_Contact( #EnMovimiento_TP1 )
   END_RUNG wire#w2
   // the same network as SCL:
   #TOut_Subir_TP(IN := "DB1_SalidasExterioresDeMesa".Mesa[#Mesa].Subir_TP_E1E3 AND #EnMovimiento_TP1 AND NOT #EstadoZona.Manual_CBx,   // "FB910_CNT_UHS"
                  R := NOT #EnMovimiento_TP1,
                  PV := #V_TOut_TP,
                  BaseUnidades_ms := "CTE_BaseUnidades_1s");
END_REGION

REGION Network 70: ERROR - TimeOut Subir TP
   RUNG wire#powerrail
      Contact( #EstadoZona.Rearme_CBx )
      S_RS(operand := #EstadoVI.Err_TOut_Subir_TP_E1_E3, s1 := #TOut_Subir_TP.QU)
      S_Coil( #EstadoVI.Error_Mx )
   END_RUNG
   // the same network as SCL:
   IF #EstadoZona.Rearme_CBx THEN
       #EstadoVI.Err_TOut_Subir_TP_E1_E3 := FALSE;   // RS flip-flop
   END_IF;
   IF #TOut_Subir_TP.QU THEN #EstadoVI.Err_TOut_Subir_TP_E1_E3 := TRUE; END_IF;
   IF #EstadoVI.Err_TOut_Subir_TP_E1_E3 THEN #EstadoVI.Error_Mx := TRUE; END_IF;
END_REGION

REGION Network 71: TMP - ERROR - TimeOut Bajar TP
   RUNG wire#powerrail
      #TOut_Bajar_TP(IN := wire#w1, R := wire#w2, PV := #V_TOut_TP, BaseUnidades_ms := "CTE_BaseUnidades_1s", QU =>, QD =>, CVU =>, CVD =>)
   END_RUNG
   RUNG wire#powerrail
      Contact( "DB1_SalidasExterioresDeMesa".Mesa[#Mesa].Bajar_TP_E1E3 )
      Contact( #EnMovimiento_TP1 )
      I_Contact( #EstadoZona.Manual_CBx )
   END_RUNG wire#w1
   RUNG wire#powerrail
      I_Contact( #EnMovimiento_TP1 )
   END_RUNG wire#w2
   // the same network as SCL:
   #TOut_Bajar_TP(IN := "DB1_SalidasExterioresDeMesa".Mesa[#Mesa].Bajar_TP_E1E3 AND #EnMovimiento_TP1 AND NOT #EstadoZona.Manual_CBx,   // "FB910_CNT_UHS"
                  R := NOT #EnMovimiento_TP1,
                  PV := #V_TOut_TP,
                  BaseUnidades_ms := "CTE_BaseUnidades_1s");
END_REGION

REGION Network 72: ERROR - TimeOut Bajar TP
   RUNG wire#powerrail
      Contact( #EstadoZona.Rearme_CBx )
      S_RS(operand := #EstadoVI.Err_TOut_Bajar_TP_E1_E3, s1 := #TOut_Bajar_TP.QU)
      S_Coil( #EstadoVI.Error_Mx )
   END_RUNG
   // the same network as SCL:
   IF #EstadoZona.Rearme_CBx THEN
       #EstadoVI.Err_TOut_Bajar_TP_E1_E3 := FALSE;   // RS flip-flop
   END_IF;
   IF #TOut_Bajar_TP.QU THEN #EstadoVI.Err_TOut_Bajar_TP_E1_E3 := TRUE; END_IF;
   IF #EstadoVI.Err_TOut_Bajar_TP_E1_E3 THEN #EstadoVI.Error_Mx := TRUE; END_IF;
END_REGION

REGION Network 73: TMP - ERROR - TimeOut Subir MQ
   RUNG wire#powerrail
      #TOut_Subir_MQ(IN := wire#w2, R := wire#w3, PV := #V_TOut_MQ, BaseUnidades_ms := "CTE_BaseUnidades_1s", QU =>, QD =>, CVU =>, CVD =>)
   END_RUNG
   RUNG wire#powerrail
      Contact( #MA_Subir_MQ1 )
      Contact( #EnMovimiento_MQ1 )
      wire#w1
      I_Contact( #EstadoZona.Manual_CBx )
   END_RUNG wire#w2
   RUNG wire#powerrail
      Contact( #MA_Subir_MQ2 )
      Contact( #EnMovimiento_MQ2 )
   END_RUNG wire#w1
   RUNG wire#powerrail
      I_Contact( #EnMovimiento_MQ1 )
      I_Contact( #EnMovimiento_MQ2 )
   END_RUNG wire#w3
   // the same network as SCL:
   #TOut_Subir_MQ(IN := ((#MA_Subir_MQ1 AND #EnMovimiento_MQ1) OR (#MA_Subir_MQ2 AND #EnMovimiento_MQ2)) AND NOT #EstadoZona.Manual_CBx,   // "FB910_CNT_UHS"
                  R := NOT #EnMovimiento_MQ1 AND NOT #EnMovimiento_MQ2,
                  PV := #V_TOut_MQ,
                  BaseUnidades_ms := "CTE_BaseUnidades_1s");
END_REGION

REGION Network 74: ERROR - TimeOut Subir MQ
   RUNG wire#powerrail
      Contact( #EstadoZona.Rearme_CBx )
      S_RS(operand := #EstadoVI.Err_TOut_Subida, s1 := #TOut_Subir_MQ.QU)
      S_Coil( #EstadoVI.Error_Mx )
   END_RUNG
   // the same network as SCL:
   IF #EstadoZona.Rearme_CBx THEN
       #EstadoVI.Err_TOut_Subida := FALSE;   // RS flip-flop
   END_IF;
   IF #TOut_Subir_MQ.QU THEN #EstadoVI.Err_TOut_Subida := TRUE; END_IF;
   IF #EstadoVI.Err_TOut_Subida THEN #EstadoVI.Error_Mx := TRUE; END_IF;
END_REGION

REGION Network 75: TMP - ERROR - TimeOut Bajar MQ
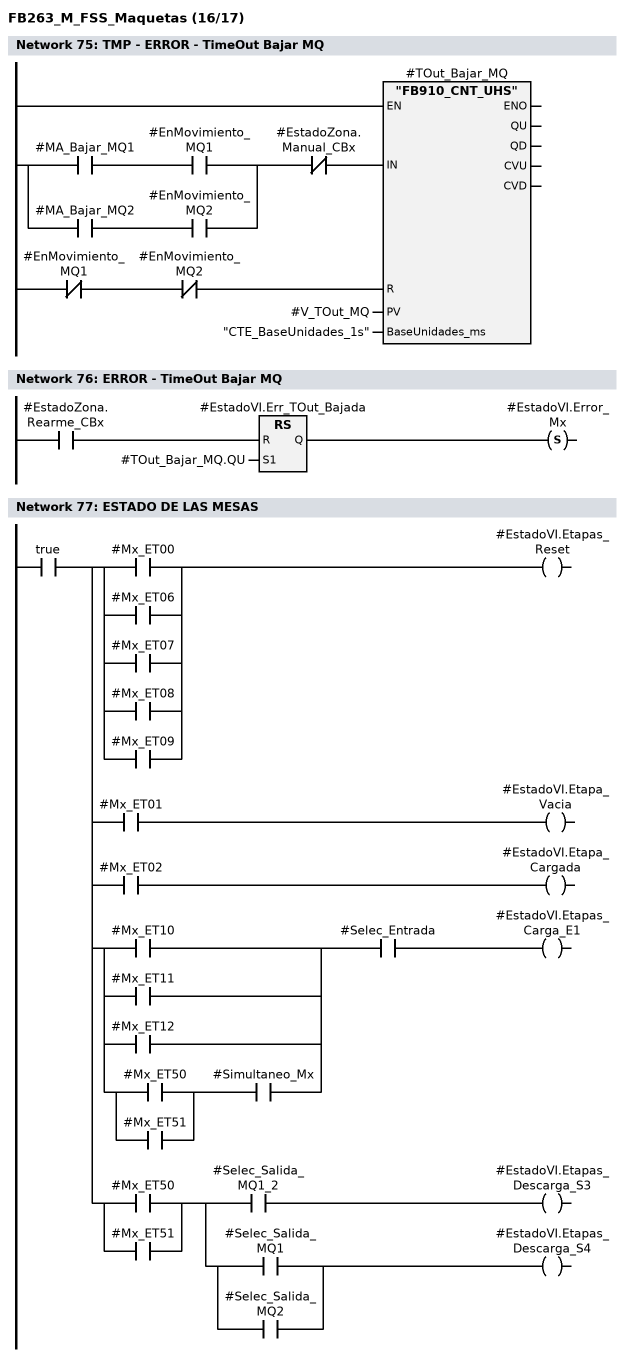
   RUNG wire#powerrail
      #TOut_Bajar_MQ(IN := wire#w2, R := wire#w3, PV := #V_TOut_MQ, BaseUnidades_ms := "CTE_BaseUnidades_1s", QU =>, QD =>, CVU =>, CVD =>)
   END_RUNG
   RUNG wire#powerrail
      Contact( #MA_Bajar_MQ1 )
      Contact( #EnMovimiento_MQ1 )
      wire#w1
      I_Contact( #EstadoZona.Manual_CBx )
   END_RUNG wire#w2
   RUNG wire#powerrail
      Contact( #MA_Bajar_MQ2 )
      Contact( #EnMovimiento_MQ2 )
   END_RUNG wire#w1
   RUNG wire#powerrail
      I_Contact( #EnMovimiento_MQ1 )
      I_Contact( #EnMovimiento_MQ2 )
   END_RUNG wire#w3
   // the same network as SCL:
   #TOut_Bajar_MQ(IN := ((#MA_Bajar_MQ1 AND #EnMovimiento_MQ1) OR (#MA_Bajar_MQ2 AND #EnMovimiento_MQ2)) AND NOT #EstadoZona.Manual_CBx,   // "FB910_CNT_UHS"
                  R := NOT #EnMovimiento_MQ1 AND NOT #EnMovimiento_MQ2,
                  PV := #V_TOut_MQ,
                  BaseUnidades_ms := "CTE_BaseUnidades_1s");
END_REGION

REGION Network 76: ERROR - TimeOut Bajar MQ
   RUNG wire#powerrail
      Contact( #EstadoZona.Rearme_CBx )
      S_RS(operand := #EstadoVI.Err_TOut_Bajada, s1 := #TOut_Bajar_MQ.QU)
      S_Coil( #EstadoVI.Error_Mx )
   END_RUNG
   // the same network as SCL:
   IF #EstadoZona.Rearme_CBx THEN
       #EstadoVI.Err_TOut_Bajada := FALSE;   // RS flip-flop
   END_IF;
   IF #TOut_Bajar_MQ.QU THEN #EstadoVI.Err_TOut_Bajada := TRUE; END_IF;
   IF #EstadoVI.Err_TOut_Bajada THEN #EstadoVI.Error_Mx := TRUE; END_IF;
END_REGION

REGION Network 77: ESTADO DE LAS MESAS
   RUNG wire#powerrail
      Contact( true )
      wire#w1
      Contact( #Mx_ET00 )
      wire#w2
      Coil( #EstadoVI.Etapas_Reset )
   END_RUNG
   RUNG wire#w1
      Contact( #Mx_ET06 )
   END_RUNG wire#w2
   RUNG wire#w1
      Contact( #Mx_ET07 )
   END_RUNG wire#w2
   RUNG wire#w1
      Contact( #Mx_ET08 )
   END_RUNG wire#w2
   RUNG wire#w1
      Contact( #Mx_ET09 )
   END_RUNG wire#w2
   RUNG wire#w1
      Contact( #Mx_ET01 )
      Coil( #EstadoVI.Etapa_Vacia )
   END_RUNG
   RUNG wire#w1
      Contact( #Mx_ET02 )
      Coil( #EstadoVI.Etapa_Cargada )
   END_RUNG
   RUNG wire#w1
      Contact( #Mx_ET10 )
      wire#w3
      Contact( #Selec_Entrada )
      Coil( #EstadoVI.Etapas_Carga_E1 )
   END_RUNG
   RUNG wire#w1
      Contact( #Mx_ET11 )
   END_RUNG wire#w3
   RUNG wire#w1
      Contact( #Mx_ET12 )
   END_RUNG wire#w3
   RUNG wire#w1
      Contact( #Mx_ET50 )
      wire#w4
      Contact( #Simultaneo_Mx )
   END_RUNG wire#w3
   RUNG wire#w1
      Contact( #Mx_ET51 )
   END_RUNG wire#w4
   RUNG wire#w1
      Contact( #Mx_ET50 )
      wire#w5
      Contact( #Selec_Salida_MQ1_2 )
      Coil( #EstadoVI.Etapas_Descarga_S3 )
   END_RUNG
   RUNG wire#w1
      Contact( #Mx_ET51 )
   END_RUNG wire#w5
   RUNG wire#w5
      Contact( #Selec_Salida_MQ1 )
      wire#w6
      Coil( #EstadoVI.Etapas_Descarga_S4 )
   END_RUNG
   RUNG wire#w5
      Contact( #Selec_Salida_MQ2 )
   END_RUNG wire#w6
   // the same network as SCL:
   #EstadoVI.Etapas_Reset := true AND (#Mx_ET00 OR #Mx_ET06 OR #Mx_ET07 OR #Mx_ET08 OR #Mx_ET09);
   #EstadoVI.Etapa_Vacia := true AND #Mx_ET01;
   #EstadoVI.Etapa_Cargada := true AND #Mx_ET02;
   #EstadoVI.Etapas_Carga_E1 := true AND (#Mx_ET10 OR #Mx_ET11 OR #Mx_ET12 OR ((#Mx_ET50 OR #Mx_ET51) AND #Simultaneo_Mx)) AND #Selec_Entrada;
   #_w1 := true AND (#Mx_ET50 OR #Mx_ET51);
   #EstadoVI.Etapas_Descarga_S3 := #_w1 AND #Selec_Salida_MQ1_2;
   #EstadoVI.Etapas_Descarga_S4 := #_w1 AND (#Selec_Salida_MQ1 OR #Selec_Salida_MQ2);
END_REGION

REGION Network 78: ENTRADAS DE LA MESA
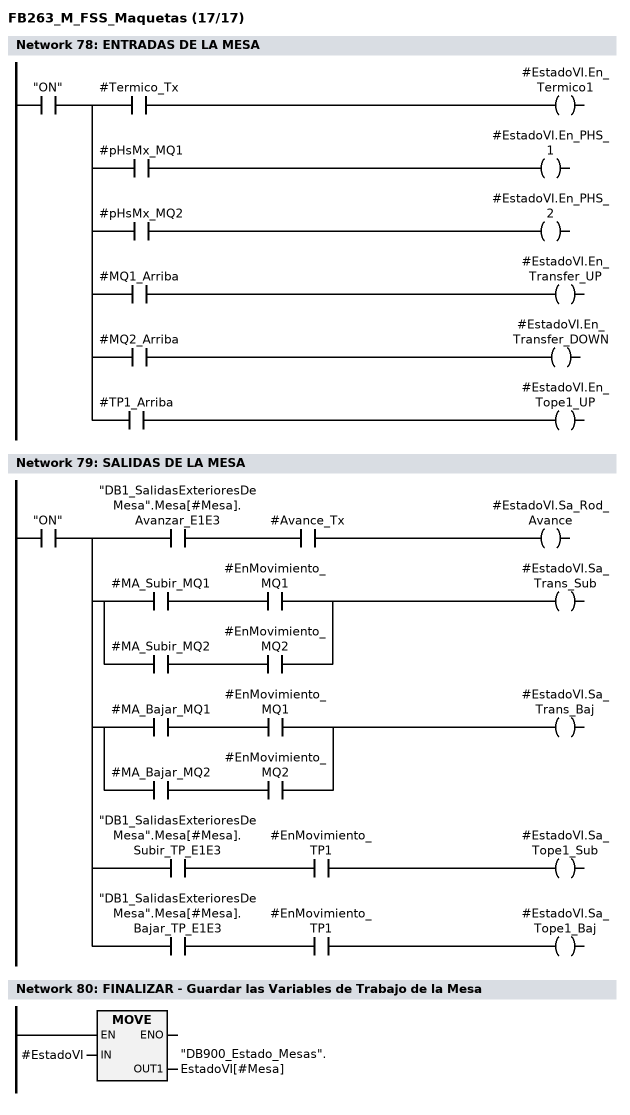
   RUNG wire#powerrail
      Contact( "ON" )
      wire#w1
      Contact( #Termico_Tx )
      Coil( #EstadoVI.En_Termico1 )
   END_RUNG
   RUNG wire#w1
      Contact( #pHsMx_MQ1 )
      Coil( #EstadoVI.En_PHS_1 )
   END_RUNG
   RUNG wire#w1
      Contact( #pHsMx_MQ2 )
      Coil( #EstadoVI.En_PHS_2 )
   END_RUNG
   RUNG wire#w1
      Contact( #MQ1_Arriba )
      Coil( #EstadoVI.En_Transfer_UP )
   END_RUNG
   RUNG wire#w1
      Contact( #MQ2_Arriba )
      Coil( #EstadoVI.En_Transfer_DOWN )
   END_RUNG
   RUNG wire#w1
      Contact( #TP1_Arriba )
      Coil( #EstadoVI.En_Tope1_UP )
   END_RUNG
   // the same network as SCL:
   #EstadoVI.En_Termico1 := "ON" AND #Termico_Tx;
   #EstadoVI.En_PHS_1 := "ON" AND #pHsMx_MQ1;
   #EstadoVI.En_PHS_2 := "ON" AND #pHsMx_MQ2;
   #EstadoVI.En_Transfer_UP := "ON" AND #MQ1_Arriba;
   #EstadoVI.En_Transfer_DOWN := "ON" AND #MQ2_Arriba;
   #EstadoVI.En_Tope1_UP := "ON" AND #TP1_Arriba;
END_REGION

REGION Network 79: SALIDAS DE LA MESA
   RUNG wire#powerrail
      Contact( "ON" )
      wire#w1
      Contact( "DB1_SalidasExterioresDeMesa".Mesa[#Mesa].Avanzar_E1E3 )
      Contact( #Avance_Tx )
      Coil( #EstadoVI.Sa_Rod_Avance )
   END_RUNG
   RUNG wire#w1
      Contact( #MA_Subir_MQ1 )
      Contact( #EnMovimiento_MQ1 )
      wire#w2
      Coil( #EstadoVI.Sa_Trans_Sub )
   END_RUNG
   RUNG wire#w1
      Contact( #MA_Subir_MQ2 )
      Contact( #EnMovimiento_MQ2 )
   END_RUNG wire#w2
   RUNG wire#w1
      Contact( #MA_Bajar_MQ1 )
      Contact( #EnMovimiento_MQ1 )
      wire#w3
      Coil( #EstadoVI.Sa_Trans_Baj )
   END_RUNG
   RUNG wire#w1
      Contact( #MA_Bajar_MQ2 )
      Contact( #EnMovimiento_MQ2 )
   END_RUNG wire#w3
   RUNG wire#w1
      Contact( "DB1_SalidasExterioresDeMesa".Mesa[#Mesa].Subir_TP_E1E3 )
      Contact( #EnMovimiento_TP1 )
      Coil( #EstadoVI.Sa_Tope1_Sub )
   END_RUNG
   RUNG wire#w1
      Contact( "DB1_SalidasExterioresDeMesa".Mesa[#Mesa].Bajar_TP_E1E3 )
      Contact( #EnMovimiento_TP1 )
      Coil( #EstadoVI.Sa_Tope1_Baj )
   END_RUNG
   // the same network as SCL:
   #EstadoVI.Sa_Rod_Avance := "ON" AND "DB1_SalidasExterioresDeMesa".Mesa[#Mesa].Avanzar_E1E3 AND #Avance_Tx;
   #EstadoVI.Sa_Trans_Sub := "ON" AND ((#MA_Subir_MQ1 AND #EnMovimiento_MQ1) OR (#MA_Subir_MQ2 AND #EnMovimiento_MQ2));
   #EstadoVI.Sa_Trans_Baj := "ON" AND ((#MA_Bajar_MQ1 AND #EnMovimiento_MQ1) OR (#MA_Bajar_MQ2 AND #EnMovimiento_MQ2));
   #EstadoVI.Sa_Tope1_Sub := "ON" AND "DB1_SalidasExterioresDeMesa".Mesa[#Mesa].Subir_TP_E1E3 AND #EnMovimiento_TP1;
   #EstadoVI.Sa_Tope1_Baj := "ON" AND "DB1_SalidasExterioresDeMesa".Mesa[#Mesa].Bajar_TP_E1E3 AND #EnMovimiento_TP1;
END_REGION

REGION Network 80: FINALIZAR - Guardar las Variables de Trabajo de la Mesa
   RUNG wire#powerrail
      Move(in := #EstadoVI, out1 => "DB900_Estado_Mesas".EstadoVI[#Mesa])
   END_RUNG
   // the same network as SCL:
   "DB900_Estado_Mesas".EstadoVI[#Mesa] := #EstadoVI;
END_REGION
END_FUNCTION_BLOCK
